ABB RAPID module: P901.mod

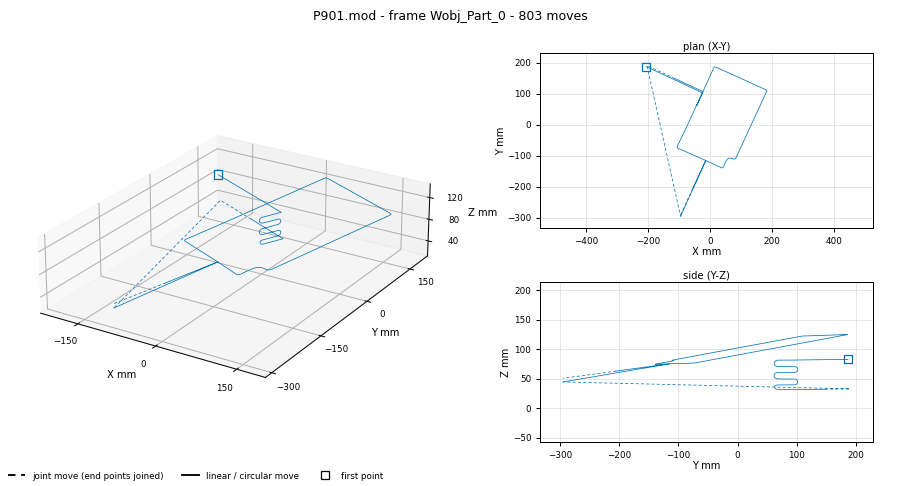
[picture p0: tool path of P901.mod in frame Wobj_Part_0, 803 of 813 moves have a stored position in this frame; points joined in program order, loops and branches not executed]
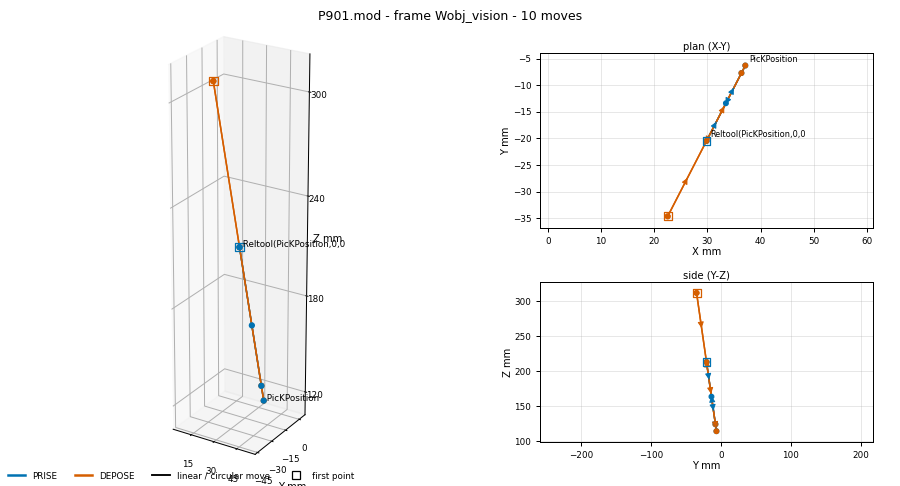
[picture p1: tool path of P901.mod in frame Wobj_vision, 10 of 813 moves have a stored position in this frame; points joined in program order, loops and branches not executed]
MODULE P901

    ! Nom         :P901
    ! Description :
    ! Créé le     :01/06/2023 14:08:14

    LOCAL CONST SPEEDDATA VitesseLente :=[3,500,0,0];
	LOCAL CONST SPEEDDATA VitesseRapide :=[30,500,0,0];
	LOCAL CONST SPEEDDATA VitesseTronconnage :=[2,500,0,0];
	LOCAL CONST SPEEDDATA VitesseTronconnageApp :=[10,500,0,0];
    !
    !Point de prise
    LOCAL PERS Robtarget PicKPosition := [[37.1247943324514,-6.27911838830437,114.674546951122],[0.0688762130874586,-0.531001244449083,0.843586238253387,0.0406940326553634],[0,0,0,0],[8.999999E+09,8.999999E+09,8.999999E+09,8.999999E+09,8.999999E+09,8.999999E+09]];
	LOCAL PERS Pose Ref := [[0,0,0],[1,0,0,0]];
    !
    !Declaration des points de meulage

    !Tr_meulage_motif_1 : Meulage d'un motif
    LOCAL CONST Robtarget Tr_meulage_motif_1_0 := [[-24.434275390625,103.0117734375,81.755546875],[0.378981302219628,-0.381323158247142,0.598057501703323,-0.594384594525059],[0,0,0,0],[8.999999E+09,8.999999E+09,8.999999E+09,8.999999E+09,8.999999E+09,8.999999E+09]];
    LOCAL CONST Robtarget Tr_meulage_motif_1_1 := [[-24.853365234375,102.103828125,81.7555625],[0.378981302219628,-0.381323158247142,0.598057501703323,-0.594384594525059],[0,0,0,0],[8.999999E+09,8.999999E+09,8.999999E+09,8.999999E+09,8.999999E+09,8.999999E+09]];
    LOCAL CONST Robtarget Tr_meulage_motif_1_2 := [[-25.27245703125,101.195890625,81.755578125],[0.378981302219628,-0.381323158247142,0.598057501703323,-0.594384594525059],[0,0,0,0],[8.999999E+09,8.999999E+09,8.999999E+09,8.999999E+09,8.999999E+09,8.999999E+09]];
    LOCAL CONST Robtarget Tr_meulage_motif_1_3 := [[-25.691546875,100.2879453125,81.75559375],[0.378981302219628,-0.381323158247142,0.598057501703323,-0.594384594525059],[0,0,0,0],[8.999999E+09,8.999999E+09,8.999999E+09,8.999999E+09,8.999999E+09,8.999999E+09]];
    LOCAL CONST Robtarget Tr_meulage_motif_1_4 := [[-26.11063671875,99.38,81.7556171875],[0.378981302219628,-0.381323158247142,0.598057501703323,-0.594384594525059],[0,0,0,0],[8.999999E+09,8.999999E+09,8.999999E+09,8.999999E+09,8.999999E+09,8.999999E+09]];
    LOCAL CONST Robtarget Tr_meulage_motif_1_5 := [[-26.5297265625,98.4720546875,81.7556328125],[0.378981302219628,-0.381323158247142,0.598057501703323,-0.594384594525059],[0,0,0,0],[8.999999E+09,8.999999E+09,8.999999E+09,8.999999E+09,8.999999E+09,8.999999E+09]];
    LOCAL CONST Robtarget Tr_meulage_motif_1_6 := [[-26.94881640625,97.564109375,81.7556484375],[0.378981302219628,-0.381323158247142,0.598057501703323,-0.594384594525059],[0,0,0,0],[8.999999E+09,8.999999E+09,8.999999E+09,8.999999E+09,8.999999E+09,8.999999E+09]];
    LOCAL CONST Robtarget Tr_meulage_motif_1_7 := [[-27.367908203125,96.6561640625,81.7556640625],[0.378981302219628,-0.381323158247142,0.598057501703323,-0.594384594525059],[0,0,0,0],[8.999999E+09,8.999999E+09,8.999999E+09,8.999999E+09,8.999999E+09,8.999999E+09]];
    LOCAL CONST Robtarget Tr_meulage_motif_1_8 := [[-27.786998046875,95.74821875,81.7556796875],[0.378981302219628,-0.381323158247142,0.598057501703323,-0.594384594525059],[0,0,0,0],[8.999999E+09,8.999999E+09,8.999999E+09,8.999999E+09,8.999999E+09,8.999999E+09]];
    LOCAL CONST Robtarget Tr_meulage_motif_1_9 := [[-28.206087890625,94.8402734375,81.7556953125],[0.378981302219628,-0.381323158247142,0.598057501703323,-0.594384594525059],[0,0,0,0],[8.999999E+09,8.999999E+09,8.999999E+09,8.999999E+09,8.999999E+09,8.999999E+09]];
    LOCAL CONST Robtarget Tr_meulage_motif_1_10 := [[-28.625177734375,93.932328125,81.7557109375],[0.378981302219628,-0.381323158247142,0.598057501703323,-0.594384594525059],[0,0,0,0],[8.999999E+09,8.999999E+09,8.999999E+09,8.999999E+09,8.999999E+09,8.999999E+09]];
    LOCAL CONST Robtarget Tr_meulage_motif_1_11 := [[-29.044267578125,93.0243828125,81.755734375],[0.378981302219628,-0.381323158247142,0.598057501703323,-0.594384594525059],[0,0,0,0],[8.999999E+09,8.999999E+09,8.999999E+09,8.999999E+09,8.999999E+09,8.999999E+09]];
    LOCAL CONST Robtarget Tr_meulage_motif_1_12 := [[-29.463359375,92.1164453125,81.75575],[0.378981302219628,-0.381323158247142,0.598057501703323,-0.594384594525059],[0,0,0,0],[8.999999E+09,8.999999E+09,8.999999E+09,8.999999E+09,8.999999E+09,8.999999E+09]];
    LOCAL CONST Robtarget Tr_meulage_motif_1_13 := [[-29.88244921875,91.2085,81.755765625],[0.378981302219628,-0.381323158247142,0.598057501703323,-0.594384594525059],[0,0,0,0],[8.999999E+09,8.999999E+09,8.999999E+09,8.999999E+09,8.999999E+09,8.999999E+09]];
    LOCAL CONST Robtarget Tr_meulage_motif_1_14 := [[-30.3015390625,90.3005546875,81.75578125],[0.378981302219628,-0.381323158247142,0.598057501703323,-0.594384594525059],[0,0,0,0],[8.999999E+09,8.999999E+09,8.999999E+09,8.999999E+09,8.999999E+09,8.999999E+09]];
    LOCAL CONST Robtarget Tr_meulage_motif_1_15 := [[-30.72062890625,89.392609375,81.755796875],[0.378981302219628,-0.381323158247142,0.598057501703323,-0.594384594525059],[0,0,0,0],[8.999999E+09,8.999999E+09,8.999999E+09,8.999999E+09,8.999999E+09,8.999999E+09]];
    LOCAL CONST Robtarget Tr_meulage_motif_1_16 := [[-31.13971875,88.4846640625,81.7558125],[0.378981302219628,-0.381323158247142,0.598057501703323,-0.594384594525059],[0,0,0,0],[8.999999E+09,8.999999E+09,8.999999E+09,8.999999E+09,8.999999E+09,8.999999E+09]];
    LOCAL CONST Robtarget Tr_meulage_motif_1_17 := [[-31.558810546875,87.57671875,81.755828125],[0.378981302219628,-0.381323158247142,0.598057501703323,-0.594384594525059],[0,0,0,0],[8.999999E+09,8.999999E+09,8.999999E+09,8.999999E+09,8.999999E+09,8.999999E+09]];
    LOCAL CONST Robtarget Tr_meulage_motif_1_18 := [[-31.977900390625,86.6687734375,81.7558515625],[0.378981302219628,-0.381323158247142,0.598057501703323,-0.594384594525059],[0,0,0,0],[8.999999E+09,8.999999E+09,8.999999E+09,8.999999E+09,8.999999E+09,8.999999E+09]];
    LOCAL CONST Robtarget Tr_meulage_motif_1_19 := [[-32.396990234375,85.760828125,81.7558671875],[0.378981302219628,-0.381323158247142,0.598057501703323,-0.594384594525059],[0,0,0,0],[8.999999E+09,8.999999E+09,8.999999E+09,8.999999E+09,8.999999E+09,8.999999E+09]];
    LOCAL CONST Robtarget Tr_meulage_motif_1_20 := [[-32.81608203125,84.8528828125,81.7558828125],[0.378981302219628,-0.381323158247142,0.598057501703323,-0.594384594525059],[0,0,0,0],[8.999999E+09,8.999999E+09,8.999999E+09,8.999999E+09,8.999999E+09,8.999999E+09]];
    LOCAL CONST Robtarget Tr_meulage_motif_1_21 := [[-33.235171875,83.9449375,81.7558984375],[0.378981302219628,-0.381323158247142,0.598057501703323,-0.594384594525059],[0,0,0,0],[8.999999E+09,8.999999E+09,8.999999E+09,8.999999E+09,8.999999E+09,8.999999E+09]];
    LOCAL CONST Robtarget Tr_meulage_motif_1_22 := [[-33.65426171875,83.0369921875,81.7559140625],[0.378981302219628,-0.381323158247142,0.598057501703323,-0.594384594525059],[0,0,0,0],[8.999999E+09,8.999999E+09,8.999999E+09,8.999999E+09,8.999999E+09,8.999999E+09]];
    LOCAL CONST Robtarget Tr_meulage_motif_1_23 := [[-34.0733515625,82.1290546875,81.7559296875],[0.378981302219628,-0.381323158247142,0.598057501703323,-0.594384594525059],[0,0,0,0],[8.999999E+09,8.999999E+09,8.999999E+09,8.999999E+09,8.999999E+09,8.999999E+09]];
    LOCAL CONST Robtarget Tr_meulage_motif_1_24 := [[-34.49244140625,81.221109375,81.755953125],[0.378981302219628,-0.381323158247142,0.598057501703323,-0.594384594525059],[0,0,0,0],[8.999999E+09,8.999999E+09,8.999999E+09,8.999999E+09,8.999999E+09,8.999999E+09]];
    LOCAL CONST Robtarget Tr_meulage_motif_1_25 := [[-34.91153125,80.3131640625,81.75596875],[0.378981302219628,-0.381323158247142,0.598057501703323,-0.594384594525059],[0,0,0,0],[8.999999E+09,8.999999E+09,8.999999E+09,8.999999E+09,8.999999E+09,8.999999E+09]];
    LOCAL CONST Robtarget Tr_meulage_motif_1_26 := [[-35.33062109375,79.40521875,81.755984375],[0.378981302219628,-0.381323158247142,0.598057501703323,-0.594384594525059],[0,0,0,0],[8.999999E+09,8.999999E+09,8.999999E+09,8.999999E+09,8.999999E+09,8.999999E+09]];
    LOCAL CONST Robtarget Tr_meulage_motif_1_27 := [[-35.7497109375,78.4972734375,81.756],[0.378981302219628,-0.381323158247142,0.598057501703323,-0.594384594525059],[0,0,0,0],[8.999999E+09,8.999999E+09,8.999999E+09,8.999999E+09,8.999999E+09,8.999999E+09]];
    LOCAL CONST Robtarget Tr_meulage_motif_1_28 := [[-36.16880078125,77.589328125,81.756015625],[0.378981302219628,-0.381323158247142,0.598057501703323,-0.594384594525059],[0,0,0,0],[8.999999E+09,8.999999E+09,8.999999E+09,8.999999E+09,8.999999E+09,8.999999E+09]];
    LOCAL CONST Robtarget Tr_meulage_motif_1_29 := [[-36.587890625,76.6813828125,81.75603125],[0.378981302219628,-0.381323158247142,0.598057501703323,-0.594384594525059],[0,0,0,0],[8.999999E+09,8.999999E+09,8.999999E+09,8.999999E+09,8.999999E+09,8.999999E+09]];
    LOCAL CONST Robtarget Tr_meulage_motif_1_30 := [[-37.006984375,75.7734375,81.756046875],[0.378981302219628,-0.381323158247142,0.598057501703323,-0.594384594525059],[0,0,0,0],[8.999999E+09,8.999999E+09,8.999999E+09,8.999999E+09,8.999999E+09,8.999999E+09]];
    LOCAL CONST Robtarget Tr_meulage_motif_1_31 := [[-37.42607421875,74.8654921875,81.7560703125],[0.378981302219628,-0.381323158247142,0.598057501703323,-0.594384594525059],[0,0,0,0],[8.999999E+09,8.999999E+09,8.999999E+09,8.999999E+09,8.999999E+09,8.999999E+09]];
    LOCAL CONST Robtarget Tr_meulage_motif_1_32 := [[-37.8451640625,73.957546875,81.7560859375],[0.378981302219628,-0.381323158247142,0.598057501703323,-0.594384594525059],[0,0,0,0],[8.999999E+09,8.999999E+09,8.999999E+09,8.999999E+09,8.999999E+09,8.999999E+09]];
    LOCAL CONST Robtarget Tr_meulage_motif_1_33 := [[-38.26425390625,73.0496015625,81.7561015625],[0.378981302219628,-0.381323158247142,0.598057501703323,-0.594384594525059],[0,0,0,0],[8.999999E+09,8.999999E+09,8.999999E+09,8.999999E+09,8.999999E+09,8.999999E+09]];
    LOCAL CONST Robtarget Tr_meulage_motif_1_34 := [[-38.68334375,72.1416640625,81.7561171875],[0.378981302219628,-0.381323158247142,0.598057501703323,-0.594384594525059],[0,0,0,0],[8.999999E+09,8.999999E+09,8.999999E+09,8.999999E+09,8.999999E+09,8.999999E+09]];
    LOCAL CONST Robtarget Tr_meulage_motif_1_35 := [[-39.10243359375,71.23371875,81.7561328125],[0.378981302219628,-0.381323158247142,0.598057501703323,-0.594384594525059],[0,0,0,0],[8.999999E+09,8.999999E+09,8.999999E+09,8.999999E+09,8.999999E+09,8.999999E+09]];
    LOCAL CONST Robtarget Tr_meulage_motif_1_36 := [[-39.5215234375,70.3257734375,81.7561484375],[0.378981302219628,-0.381323158247142,0.598057501703323,-0.594384594525059],[0,0,0,0],[8.999999E+09,8.999999E+09,8.999999E+09,8.999999E+09,8.999999E+09,8.999999E+09]];
    LOCAL CONST Robtarget Tr_meulage_motif_1_37 := [[-39.94061328125,69.417828125,81.7561640625],[0.378981302219628,-0.381323158247142,0.598057501703323,-0.594384594525059],[0,0,0,0],[8.999999E+09,8.999999E+09,8.999999E+09,8.999999E+09,8.999999E+09,8.999999E+09]];
    LOCAL CONST Robtarget Tr_meulage_motif_1_38 := [[-40.359703125,68.5098828125,81.7561875],[0.378981302219628,-0.381323158247142,0.598057501703323,-0.594384594525059],[0,0,0,0],[8.999999E+09,8.999999E+09,8.999999E+09,8.999999E+09,8.999999E+09,8.999999E+09]];
    LOCAL CONST Robtarget Tr_meulage_motif_1_39 := [[-40.77410546875,67.6079609375,81.6456171875],[0.378981302219628,-0.381323158247142,0.598057501703323,-0.594384594525059],[0,0,0,0],[8.999999E+09,8.999999E+09,8.999999E+09,8.999999E+09,8.999999E+09,8.999999E+09]];
    LOCAL CONST Robtarget Tr_meulage_motif_1_40 := [[-41.16776953125,66.747203125,81.4344765625],[0.378981302219628,-0.381323158247142,0.598057501703323,-0.594384594525059],[0,0,0,0],[8.999999E+09,8.999999E+09,8.999999E+09,8.999999E+09,8.999999E+09,8.999999E+09]];
    LOCAL CONST Robtarget Tr_meulage_motif_1_41 := [[-41.52126953125,65.9711953125,81.1626796875],[0.378981302219628,-0.381323158247142,0.598057501703323,-0.594384594525059],[0,0,0,0],[8.999999E+09,8.999999E+09,8.999999E+09,8.999999E+09,8.999999E+09,8.999999E+09]];
    LOCAL CONST Robtarget Tr_meulage_motif_1_42 := [[-41.83163671875,65.28847265625,80.8867890625],[0.378981302219628,-0.381323158247142,0.598057501703323,-0.594384594525059],[0,0,0,0],[8.999999E+09,8.999999E+09,8.999999E+09,8.999999E+09,8.999999E+09,8.999999E+09]];
    LOCAL CONST Robtarget Tr_meulage_motif_1_43 := [[-42.2843203125,64.28471484375,80.2707578125],[0.378981302219628,-0.381323158247142,0.598057501703323,-0.594384594525059],[0,0,0,0],[8.999999E+09,8.999999E+09,8.999999E+09,8.999999E+09,8.999999E+09,8.999999E+09]];
    LOCAL CONST Robtarget Tr_meulage_motif_1_44 := [[-42.701359375,63.34951171875,79.42321875],[0.378981302219628,-0.381323158247142,0.598057501703323,-0.594384594525059],[0,0,0,0],[8.999999E+09,8.999999E+09,8.999999E+09,8.999999E+09,8.999999E+09,8.999999E+09]];
    LOCAL CONST Robtarget Tr_meulage_motif_1_45 := [[-43.04204296875,62.5731484375,78.399484375],[0.378981302219628,-0.381323158247142,0.598057501703323,-0.594384594525059],[0,0,0,0],[8.999999E+09,8.999999E+09,8.999999E+09,8.999999E+09,8.999999E+09,8.999999E+09]];
    LOCAL CONST Robtarget Tr_meulage_motif_1_46 := [[-43.23075,62.122578125,77.2834453125],[0.378981302219628,-0.381323158247142,0.598057501703323,-0.594384594525059],[0,0,0,0],[8.999999E+09,8.999999E+09,8.999999E+09,8.999999E+09,8.999999E+09,8.999999E+09]];
    LOCAL CONST Robtarget Tr_meulage_motif_1_47 := [[-43.2321953125,62.09342578125,76.5875625],[0.378981302219628,-0.381323158247142,0.598057501703323,-0.594384594525059],[0,0,0,0],[8.999999E+09,8.999999E+09,8.999999E+09,8.999999E+09,8.999999E+09,8.999999E+09]];
    LOCAL CONST Robtarget Tr_meulage_motif_1_48 := [[-43.2227890625,62.08907421875,75.926390625],[0.378981302219628,-0.381323158247142,0.598057501703323,-0.594384594525059],[0,0,0,0],[8.999999E+09,8.999999E+09,8.999999E+09,8.999999E+09,8.999999E+09,8.999999E+09]];
    LOCAL CONST Robtarget Tr_meulage_motif_1_49 := [[-43.190390625,62.134546875,75.2653828125],[0.378981302219628,-0.381323158247142,0.598057501703323,-0.594384594525059],[0,0,0,0],[8.999999E+09,8.999999E+09,8.999999E+09,8.999999E+09,8.999999E+09,8.999999E+09]];
    LOCAL CONST Robtarget Tr_meulage_motif_1_50 := [[-42.965921875,62.5796484375,74.1637578125],[0.378981302219628,-0.381323158247142,0.598057501703323,-0.594384594525059],[0,0,0,0],[8.999999E+09,8.999999E+09,8.999999E+09,8.999999E+09,8.999999E+09,8.999999E+09]];
    LOCAL CONST Robtarget Tr_meulage_motif_1_51 := [[-42.59260546875,63.3507890625,73.1572421875],[0.378981302219628,-0.381323158247142,0.598057501703323,-0.594384594525059],[0,0,0,0],[8.999999E+09,8.999999E+09,8.999999E+09,8.999999E+09,8.999999E+09,8.999999E+09]];
    LOCAL CONST Robtarget Tr_meulage_motif_1_52 := [[-42.15191796875,64.27452734375,72.328453125],[0.378981302219628,-0.381323158247142,0.598057501703323,-0.594384594525059],[0,0,0,0],[8.999999E+09,8.999999E+09,8.999999E+09,8.999999E+09,8.999999E+09,8.999999E+09]];
    LOCAL CONST Robtarget Tr_meulage_motif_1_53 := [[-41.85833203125,64.895765625,71.932734375],[0.378981302219628,-0.381323158247142,0.598057501703323,-0.594384594525059],[0,0,0,0],[8.999999E+09,8.999999E+09,8.999999E+09,8.999999E+09,8.999999E+09,8.999999E+09]];
    LOCAL CONST Robtarget Tr_meulage_motif_1_54 := [[-41.36602734375,65.9441015625,71.44525],[0.378981302219628,-0.381323158247142,0.598057501703323,-0.594384594525059],[0,0,0,0],[8.999999E+09,8.999999E+09,8.999999E+09,8.999999E+09,8.999999E+09,8.999999E+09]];
    LOCAL CONST Robtarget Tr_meulage_motif_1_55 := [[-41.00812890625,66.7096015625,71.181171875],[0.378981302219628,-0.381323158247142,0.598057501703323,-0.594384594525059],[0,0,0,0],[8.999999E+09,8.999999E+09,8.999999E+09,8.999999E+09,8.999999E+09,8.999999E+09]];
    LOCAL CONST Robtarget Tr_meulage_motif_1_56 := [[-40.61462890625,67.5544609375,70.9767109375],[0.378981302219628,-0.381323158247142,0.598057501703323,-0.594384594525059],[0,0,0,0],[8.999999E+09,8.999999E+09,8.999999E+09,8.999999E+09,8.999999E+09,8.999999E+09]];
    LOCAL CONST Robtarget Tr_meulage_motif_1_57 := [[-40.20171875,68.444953125,70.8681171875],[0.378981302219628,-0.381323158247142,0.598057501703323,-0.594384594525059],[0,0,0,0],[8.999999E+09,8.999999E+09,8.999999E+09,8.999999E+09,8.999999E+09,8.999999E+09]];
    LOCAL CONST Robtarget Tr_meulage_motif_1_58 := [[-39.78417578125,69.3454140625,70.757515625],[0.378981302219628,-0.381323158247142,0.598057501703323,-0.594384594525059],[0,0,0,0],[8.999999E+09,8.999999E+09,8.999999E+09,8.999999E+09,8.999999E+09,8.999999E+09]];
    LOCAL CONST Robtarget Tr_meulage_motif_1_59 := [[-39.3650859375,70.253359375,70.7575],[0.378981302219628,-0.381323158247142,0.598057501703323,-0.594384594525059],[0,0,0,0],[8.999999E+09,8.999999E+09,8.999999E+09,8.999999E+09,8.999999E+09,8.999999E+09]];
    LOCAL CONST Robtarget Tr_meulage_motif_1_60 := [[-38.9459921875,71.1613046875,70.757484375],[0.378981302219628,-0.381323158247142,0.598057501703323,-0.594384594525059],[0,0,0,0],[8.999999E+09,8.999999E+09,8.999999E+09,8.999999E+09,8.999999E+09,8.999999E+09]];
    LOCAL CONST Robtarget Tr_meulage_motif_1_61 := [[-38.52690234375,72.06925,70.75746875],[0.378981302219628,-0.381323158247142,0.598057501703323,-0.594384594525059],[0,0,0,0],[8.999999E+09,8.999999E+09,8.999999E+09,8.999999E+09,8.999999E+09,8.999999E+09]];
    LOCAL CONST Robtarget Tr_meulage_motif_1_62 := [[-38.1078125,72.9771953125,70.757453125],[0.378981302219628,-0.381323158247142,0.598057501703323,-0.594384594525059],[0,0,0,0],[8.999999E+09,8.999999E+09,8.999999E+09,8.999999E+09,8.999999E+09,8.999999E+09]];
    LOCAL CONST Robtarget Tr_meulage_motif_1_63 := [[-37.68872265625,73.8851328125,70.7574375],[0.378981302219628,-0.381323158247142,0.598057501703323,-0.594384594525059],[0,0,0,0],[8.999999E+09,8.999999E+09,8.999999E+09,8.999999E+09,8.999999E+09,8.999999E+09]];
    LOCAL CONST Robtarget Tr_meulage_motif_1_64 := [[-37.2696328125,74.793078125,70.7574140625],[0.378981302219628,-0.381323158247142,0.598057501703323,-0.594384594525059],[0,0,0,0],[8.999999E+09,8.999999E+09,8.999999E+09,8.999999E+09,8.999999E+09,8.999999E+09]];
    LOCAL CONST Robtarget Tr_meulage_motif_1_65 := [[-36.85054296875,75.7010234375,70.7573984375],[0.378981302219628,-0.381323158247142,0.598057501703323,-0.594384594525059],[0,0,0,0],[8.999999E+09,8.999999E+09,8.999999E+09,8.999999E+09,8.999999E+09,8.999999E+09]];
    LOCAL CONST Robtarget Tr_meulage_motif_1_66 := [[-36.431453125,76.60896875,70.7573828125],[0.378981302219628,-0.381323158247142,0.598057501703323,-0.594384594525059],[0,0,0,0],[8.999999E+09,8.999999E+09,8.999999E+09,8.999999E+09,8.999999E+09,8.999999E+09]];
    LOCAL CONST Robtarget Tr_meulage_motif_1_67 := [[-36.01236328125,77.5169140625,70.7573671875],[0.378981302219628,-0.381323158247142,0.598057501703323,-0.594384594525059],[0,0,0,0],[8.999999E+09,8.999999E+09,8.999999E+09,8.999999E+09,8.999999E+09,8.999999E+09]];
    LOCAL CONST Robtarget Tr_meulage_motif_1_68 := [[-35.5932734375,78.424859375,70.7573515625],[0.378981302219628,-0.381323158247142,0.598057501703323,-0.594384594525059],[0,0,0,0],[8.999999E+09,8.999999E+09,8.999999E+09,8.999999E+09,8.999999E+09,8.999999E+09]];
    LOCAL CONST Robtarget Tr_meulage_motif_1_69 := [[-35.17418359375,79.3328046875,70.7573359375],[0.378981302219628,-0.381323158247142,0.598057501703323,-0.594384594525059],[0,0,0,0],[8.999999E+09,8.999999E+09,8.999999E+09,8.999999E+09,8.999999E+09,8.999999E+09]];
    LOCAL CONST Robtarget Tr_meulage_motif_1_70 := [[-34.75508984375,80.24075,70.7573203125],[0.378981302219628,-0.381323158247142,0.598057501703323,-0.594384594525059],[0,0,0,0],[8.999999E+09,8.999999E+09,8.999999E+09,8.999999E+09,8.999999E+09,8.999999E+09]];
    LOCAL CONST Robtarget Tr_meulage_motif_1_71 := [[-34.336,81.1486953125,70.757296875],[0.378981302219628,-0.381323158247142,0.598057501703323,-0.594384594525059],[0,0,0,0],[8.999999E+09,8.999999E+09,8.999999E+09,8.999999E+09,8.999999E+09,8.999999E+09]];
    LOCAL CONST Robtarget Tr_meulage_motif_1_72 := [[-33.91691015625,82.056640625,70.75728125],[0.378981302219628,-0.381323158247142,0.598057501703323,-0.594384594525059],[0,0,0,0],[8.999999E+09,8.999999E+09,8.999999E+09,8.999999E+09,8.999999E+09,8.999999E+09]];
    LOCAL CONST Robtarget Tr_meulage_motif_1_73 := [[-33.4978203125,82.9645859375,70.757265625],[0.378981302219628,-0.381323158247142,0.598057501703323,-0.594384594525059],[0,0,0,0],[8.999999E+09,8.999999E+09,8.999999E+09,8.999999E+09,8.999999E+09,8.999999E+09]];
    LOCAL CONST Robtarget Tr_meulage_motif_1_74 := [[-33.07873046875,83.8725234375,70.75725],[0.378981302219628,-0.381323158247142,0.598057501703323,-0.594384594525059],[0,0,0,0],[8.999999E+09,8.999999E+09,8.999999E+09,8.999999E+09,8.999999E+09,8.999999E+09]];
    LOCAL CONST Robtarget Tr_meulage_motif_1_75 := [[-32.659640625,84.78046875,70.757234375],[0.378981302219628,-0.381323158247142,0.598057501703323,-0.594384594525059],[0,0,0,0],[8.999999E+09,8.999999E+09,8.999999E+09,8.999999E+09,8.999999E+09,8.999999E+09]];
    LOCAL CONST Robtarget Tr_meulage_motif_1_76 := [[-32.24055078125,85.6884140625,70.75721875],[0.378981302219628,-0.381323158247142,0.598057501703323,-0.594384594525059],[0,0,0,0],[8.999999E+09,8.999999E+09,8.999999E+09,8.999999E+09,8.999999E+09,8.999999E+09]];
    LOCAL CONST Robtarget Tr_meulage_motif_1_77 := [[-31.821458984375,86.596359375,70.757203125],[0.378981302219628,-0.381323158247142,0.598057501703323,-0.594384594525059],[0,0,0,0],[8.999999E+09,8.999999E+09,8.999999E+09,8.999999E+09,8.999999E+09,8.999999E+09]];
    LOCAL CONST Robtarget Tr_meulage_motif_1_78 := [[-31.402369140625,87.5043046875,70.7571796875],[0.378981302219628,-0.381323158247142,0.598057501703323,-0.594384594525059],[0,0,0,0],[8.999999E+09,8.999999E+09,8.999999E+09,8.999999E+09,8.999999E+09,8.999999E+09]];
    LOCAL CONST Robtarget Tr_meulage_motif_1_79 := [[-30.983279296875,88.41225,70.7571640625],[0.378981302219628,-0.381323158247142,0.598057501703323,-0.594384594525059],[0,0,0,0],[8.999999E+09,8.999999E+09,8.999999E+09,8.999999E+09,8.999999E+09,8.999999E+09]];
    LOCAL CONST Robtarget Tr_meulage_motif_1_80 := [[-30.564189453125,89.3201953125,70.7571484375],[0.378981302219628,-0.381323158247142,0.598057501703323,-0.594384594525059],[0,0,0,0],[8.999999E+09,8.999999E+09,8.999999E+09,8.999999E+09,8.999999E+09,8.999999E+09]];
    LOCAL CONST Robtarget Tr_meulage_motif_1_81 := [[-30.145099609375,90.228140625,70.7571328125],[0.378981302219628,-0.381323158247142,0.598057501703323,-0.594384594525059],[0,0,0,0],[8.999999E+09,8.999999E+09,8.999999E+09,8.999999E+09,8.999999E+09,8.999999E+09]];
    LOCAL CONST Robtarget Tr_meulage_motif_1_82 := [[-29.7260078125,91.1360859375,70.7571171875],[0.378981302219628,-0.381323158247142,0.598057501703323,-0.594384594525059],[0,0,0,0],[8.999999E+09,8.999999E+09,8.999999E+09,8.999999E+09,8.999999E+09,8.999999E+09]];
    LOCAL CONST Robtarget Tr_meulage_motif_1_83 := [[-29.30691796875,92.04403125,70.7571015625],[0.378981302219628,-0.381323158247142,0.598057501703323,-0.594384594525059],[0,0,0,0],[8.999999E+09,8.999999E+09,8.999999E+09,8.999999E+09,8.999999E+09,8.999999E+09]];
    LOCAL CONST Robtarget Tr_meulage_motif_1_84 := [[-28.887828125,92.9519765625,70.7570859375],[0.378981302219628,-0.381323158247142,0.598057501703323,-0.594384594525059],[0,0,0,0],[8.999999E+09,8.999999E+09,8.999999E+09,8.999999E+09,8.999999E+09,8.999999E+09]];
    LOCAL CONST Robtarget Tr_meulage_motif_1_85 := [[-28.46873828125,93.8599140625,70.7570625],[0.378981302219628,-0.381323158247142,0.598057501703323,-0.594384594525059],[0,0,0,0],[8.999999E+09,8.999999E+09,8.999999E+09,8.999999E+09,8.999999E+09,8.999999E+09]];
    LOCAL CONST Robtarget Tr_meulage_motif_1_86 := [[-28.0496484375,94.767859375,70.757046875],[0.378981302219628,-0.381323158247142,0.598057501703323,-0.594384594525059],[0,0,0,0],[8.999999E+09,8.999999E+09,8.999999E+09,8.999999E+09,8.999999E+09,8.999999E+09]];
    LOCAL CONST Robtarget Tr_meulage_motif_1_87 := [[-27.63055859375,95.6758046875,70.75703125],[0.378981302219628,-0.381323158247142,0.598057501703323,-0.594384594525059],[0,0,0,0],[8.999999E+09,8.999999E+09,8.999999E+09,8.999999E+09,8.999999E+09,8.999999E+09]];
    LOCAL CONST Robtarget Tr_meulage_motif_1_88 := [[-27.211466796875,96.58375,70.757015625],[0.378981302219628,-0.381323158247142,0.598057501703323,-0.594384594525059],[0,0,0,0],[8.999999E+09,8.999999E+09,8.999999E+09,8.999999E+09,8.999999E+09,8.999999E+09]];
    LOCAL CONST Robtarget Tr_meulage_motif_1_89 := [[-26.793921875,97.48421875,70.646421875],[0.378981302219628,-0.381323158247142,0.598057501703323,-0.594384594525059],[0,0,0,0],[8.999999E+09,8.999999E+09,8.999999E+09,8.999999E+09,8.999999E+09,8.999999E+09]];
    LOCAL CONST Robtarget Tr_meulage_motif_1_90 := [[-26.394248046875,98.3421953125,70.4352421875],[0.378981302219628,-0.381323158247142,0.598057501703323,-0.594384594525059],[0,0,0,0],[8.999999E+09,8.999999E+09,8.999999E+09,8.999999E+09,8.999999E+09,8.999999E+09]];
    LOCAL CONST Robtarget Tr_meulage_motif_1_91 := [[-26.033017578125,99.114625,70.1634140625],[0.378981302219628,-0.381323158247142,0.598057501703323,-0.594384594525059],[0,0,0,0],[8.999999E+09,8.999999E+09,8.999999E+09,8.999999E+09,8.999999E+09,8.999999E+09]];
    LOCAL CONST Robtarget Tr_meulage_motif_1_92 := [[-25.7305078125,99.758625,69.8592890625],[0.378981302219628,-0.381323158247142,0.598057501703323,-0.594384594525059],[0,0,0,0],[8.999999E+09,8.999999E+09,8.999999E+09,8.999999E+09,8.999999E+09,8.999999E+09]];
    LOCAL CONST Robtarget Tr_meulage_motif_1_93 := [[-25.28755078125,100.6935078125,69.1968203125],[0.378981302219628,-0.381323158247142,0.598057501703323,-0.594384594525059],[0,0,0,0],[8.999999E+09,8.999999E+09,8.999999E+09,8.999999E+09,8.999999E+09,8.999999E+09]];
    LOCAL CONST Robtarget Tr_meulage_motif_1_94 := [[-24.89673046875,101.5064765625,68.2949765625],[0.378981302219628,-0.381323158247142,0.598057501703323,-0.594384594525059],[0,0,0,0],[8.999999E+09,8.999999E+09,8.999999E+09,8.999999E+09,8.999999E+09,8.999999E+09]];
    LOCAL CONST Robtarget Tr_meulage_motif_1_95 := [[-24.65765234375,101.9853125,67.2490625],[0.378981302219628,-0.381323158247142,0.598057501703323,-0.594384594525059],[0,0,0,0],[8.999999E+09,8.999999E+09,8.999999E+09,8.999999E+09,8.999999E+09,8.999999E+09]];
    LOCAL CONST Robtarget Tr_meulage_motif_1_96 := [[-24.570353515625,102.1485234375,66.5559296875],[0.378981302219628,-0.381323158247142,0.598057501703323,-0.594384594525059],[0,0,0,0],[8.999999E+09,8.999999E+09,8.999999E+09,8.999999E+09,8.999999E+09,8.999999E+09]];
    LOCAL CONST Robtarget Tr_meulage_motif_1_97 := [[-24.532646484375,102.201421875,65.7860234375],[0.378981302219628,-0.381323158247142,0.598057501703323,-0.594384594525059],[0,0,0,0],[8.999999E+09,8.999999E+09,8.999999E+09,8.999999E+09,8.999999E+09,8.999999E+09]];
    LOCAL CONST Robtarget Tr_meulage_motif_1_98 := [[-24.549751953125,102.135578125,65.0162421875],[0.378981302219628,-0.381323158247142,0.598057501703323,-0.594384594525059],[0,0,0,0],[8.999999E+09,8.999999E+09,8.999999E+09,8.999999E+09,8.999999E+09,8.999999E+09]];
    LOCAL CONST Robtarget Tr_meulage_motif_1_99 := [[-24.709837890625,101.7473125,63.90813671875],[0.378981302219628,-0.381323158247142,0.598057501703323,-0.594384594525059],[0,0,0,0],[8.999999E+09,8.999999E+09,8.999999E+09,8.999999E+09,8.999999E+09,8.999999E+09]];
    LOCAL CONST Robtarget Tr_meulage_motif_1_100 := [[-24.875142578125,101.36728125,63.32252734375],[0.378981302219628,-0.381323158247142,0.598057501703323,-0.594384594525059],[0,0,0,0],[8.999999E+09,8.999999E+09,8.999999E+09,8.999999E+09,8.999999E+09,8.999999E+09]];
    LOCAL CONST Robtarget Tr_meulage_motif_1_101 := [[-25.234310546875,100.555984375,62.4355234375],[0.378981302219628,-0.381323158247142,0.598057501703323,-0.594384594525059],[0,0,0,0],[8.999999E+09,8.999999E+09,8.999999E+09,8.999999E+09,8.999999E+09,8.999999E+09]];
    LOCAL CONST Robtarget Tr_meulage_motif_1_102 := [[-25.473875,100.021484375,62.0212734375],[0.378981302219628,-0.381323158247142,0.598057501703323,-0.594384594525059],[0,0,0,0],[8.999999E+09,8.999999E+09,8.999999E+09,8.999999E+09,8.999999E+09,8.999999E+09]];
    LOCAL CONST Robtarget Tr_meulage_motif_1_103 := [[-25.934640625,99.00290625,61.477265625],[0.378981302219628,-0.381323158247142,0.598057501703323,-0.594384594525059],[0,0,0,0],[8.999999E+09,8.999999E+09,8.999999E+09,8.999999E+09,8.999999E+09,8.999999E+09]];
    LOCAL CONST Robtarget Tr_meulage_motif_1_104 := [[-26.276435546875,98.2513671875,61.18181640625],[0.378981302219628,-0.381323158247142,0.598057501703323,-0.594384594525059],[0,0,0,0],[8.999999E+09,8.999999E+09,8.999999E+09,8.999999E+09,8.999999E+09,8.999999E+09]];
    LOCAL CONST Robtarget Tr_meulage_motif_1_105 := [[-26.66412109375,97.4038125,60.97738671875],[0.378981302219628,-0.381323158247142,0.598057501703323,-0.594384594525059],[0,0,0,0],[8.999999E+09,8.999999E+09,8.999999E+09,8.999999E+09,8.999999E+09,8.999999E+09]];
    LOCAL CONST Robtarget Tr_meulage_motif_1_106 := [[-27.073939453125,96.5118984375,60.86882421875],[0.378981302219628,-0.381323158247142,0.598057501703323,-0.594384594525059],[0,0,0,0],[8.999999E+09,8.999999E+09,8.999999E+09,8.999999E+09,8.999999E+09,8.999999E+09]];
    LOCAL CONST Robtarget Tr_meulage_motif_1_107 := [[-27.48833984375,95.6099765625,60.7582578125],[0.378981302219628,-0.381323158247142,0.598057501703323,-0.594384594525059],[0,0,0,0],[8.999999E+09,8.999999E+09,8.999999E+09,8.999999E+09,8.999999E+09,8.999999E+09]];
    LOCAL CONST Robtarget Tr_meulage_motif_1_108 := [[-27.9074296875,94.70203125,60.75827734375],[0.378981302219628,-0.381323158247142,0.598057501703323,-0.594384594525059],[0,0,0,0],[8.999999E+09,8.999999E+09,8.999999E+09,8.999999E+09,8.999999E+09,8.999999E+09]];
    LOCAL CONST Robtarget Tr_meulage_motif_1_109 := [[-28.32651953125,93.7940859375,60.75829296875],[0.378981302219628,-0.381323158247142,0.598057501703323,-0.594384594525059],[0,0,0,0],[8.999999E+09,8.999999E+09,8.999999E+09,8.999999E+09,8.999999E+09,8.999999E+09]];
    LOCAL CONST Robtarget Tr_meulage_motif_1_110 := [[-28.745609375,92.886140625,60.75830859375],[0.378981302219628,-0.381323158247142,0.598057501703323,-0.594384594525059],[0,0,0,0],[8.999999E+09,8.999999E+09,8.999999E+09,8.999999E+09,8.999999E+09,8.999999E+09]];
    LOCAL CONST Robtarget Tr_meulage_motif_1_111 := [[-29.164701171875,91.9781953125,60.758328125],[0.378981302219628,-0.381323158247142,0.598057501703323,-0.594384594525059],[0,0,0,0],[8.999999E+09,8.999999E+09,8.999999E+09,8.999999E+09,8.999999E+09,8.999999E+09]];
    LOCAL CONST Robtarget Tr_meulage_motif_1_112 := [[-29.583791015625,91.0702578125,60.75834375],[0.378981302219628,-0.381323158247142,0.598057501703323,-0.594384594525059],[0,0,0,0],[8.999999E+09,8.999999E+09,8.999999E+09,8.999999E+09,8.999999E+09,8.999999E+09]];
    LOCAL CONST Robtarget Tr_meulage_motif_1_113 := [[-30.002880859375,90.1623125,60.758359375],[0.378981302219628,-0.381323158247142,0.598057501703323,-0.594384594525059],[0,0,0,0],[8.999999E+09,8.999999E+09,8.999999E+09,8.999999E+09,8.999999E+09,8.999999E+09]];
    LOCAL CONST Robtarget Tr_meulage_motif_1_114 := [[-30.421970703125,89.2543671875,60.75837890625],[0.378981302219628,-0.381323158247142,0.598057501703323,-0.594384594525059],[0,0,0,0],[8.999999E+09,8.999999E+09,8.999999E+09,8.999999E+09,8.999999E+09,8.999999E+09]];
    LOCAL CONST Robtarget Tr_meulage_motif_1_115 := [[-30.841060546875,88.346421875,60.75839453125],[0.378981302219628,-0.381323158247142,0.598057501703323,-0.594384594525059],[0,0,0,0],[8.999999E+09,8.999999E+09,8.999999E+09,8.999999E+09,8.999999E+09,8.999999E+09]];
    LOCAL CONST Robtarget Tr_meulage_motif_1_116 := [[-31.26015234375,87.4384765625,60.75841015625],[0.378981302219628,-0.381323158247142,0.598057501703323,-0.594384594525059],[0,0,0,0],[8.999999E+09,8.999999E+09,8.999999E+09,8.999999E+09,8.999999E+09,8.999999E+09]];
    LOCAL CONST Robtarget Tr_meulage_motif_1_117 := [[-31.6792421875,86.53053125,60.75842578125],[0.378981302219628,-0.381323158247142,0.598057501703323,-0.594384594525059],[0,0,0,0],[8.999999E+09,8.999999E+09,8.999999E+09,8.999999E+09,8.999999E+09,8.999999E+09]];
    LOCAL CONST Robtarget Tr_meulage_motif_1_118 := [[-32.09833203125,85.6225859375,60.7584453125],[0.378981302219628,-0.381323158247142,0.598057501703323,-0.594384594525059],[0,0,0,0],[8.999999E+09,8.999999E+09,8.999999E+09,8.999999E+09,8.999999E+09,8.999999E+09]];
    LOCAL CONST Robtarget Tr_meulage_motif_1_119 := [[-32.517421875,84.714640625,60.7584609375],[0.378981302219628,-0.381323158247142,0.598057501703323,-0.594384594525059],[0,0,0,0],[8.999999E+09,8.999999E+09,8.999999E+09,8.999999E+09,8.999999E+09,8.999999E+09]];
    LOCAL CONST Robtarget Tr_meulage_motif_1_120 := [[-32.93651171875,83.8066953125,60.7584765625],[0.378981302219628,-0.381323158247142,0.598057501703323,-0.594384594525059],[0,0,0,0],[8.999999E+09,8.999999E+09,8.999999E+09,8.999999E+09,8.999999E+09,8.999999E+09]];
    LOCAL CONST Robtarget Tr_meulage_motif_1_121 := [[-33.3556015625,82.89875,60.75849609375],[0.378981302219628,-0.381323158247142,0.598057501703323,-0.594384594525059],[0,0,0,0],[8.999999E+09,8.999999E+09,8.999999E+09,8.999999E+09,8.999999E+09,8.999999E+09]];
    LOCAL CONST Robtarget Tr_meulage_motif_1_122 := [[-33.77469140625,81.9908046875,60.75851171875],[0.378981302219628,-0.381323158247142,0.598057501703323,-0.594384594525059],[0,0,0,0],[8.999999E+09,8.999999E+09,8.999999E+09,8.999999E+09,8.999999E+09,8.999999E+09]];
    LOCAL CONST Robtarget Tr_meulage_motif_1_123 := [[-34.19378125,81.0828671875,60.75852734375],[0.378981302219628,-0.381323158247142,0.598057501703323,-0.594384594525059],[0,0,0,0],[8.999999E+09,8.999999E+09,8.999999E+09,8.999999E+09,8.999999E+09,8.999999E+09]];
    LOCAL CONST Robtarget Tr_meulage_motif_1_124 := [[-34.612875,80.174921875,60.758546875],[0.378981302219628,-0.381323158247142,0.598057501703323,-0.594384594525059],[0,0,0,0],[8.999999E+09,8.999999E+09,8.999999E+09,8.999999E+09,8.999999E+09,8.999999E+09]];
    LOCAL CONST Robtarget Tr_meulage_motif_1_125 := [[-35.03196484375,79.2669765625,60.7585625],[0.378981302219628,-0.381323158247142,0.598057501703323,-0.594384594525059],[0,0,0,0],[8.999999E+09,8.999999E+09,8.999999E+09,8.999999E+09,8.999999E+09,8.999999E+09]];
    LOCAL CONST Robtarget Tr_meulage_motif_1_126 := [[-35.4510546875,78.35903125,60.758578125],[0.378981302219628,-0.381323158247142,0.598057501703323,-0.594384594525059],[0,0,0,0],[8.999999E+09,8.999999E+09,8.999999E+09,8.999999E+09,8.999999E+09,8.999999E+09]];
    LOCAL CONST Robtarget Tr_meulage_motif_1_127 := [[-35.87014453125,77.4510859375,60.75859375],[0.378981302219628,-0.381323158247142,0.598057501703323,-0.594384594525059],[0,0,0,0],[8.999999E+09,8.999999E+09,8.999999E+09,8.999999E+09,8.999999E+09,8.999999E+09]];
    LOCAL CONST Robtarget Tr_meulage_motif_1_128 := [[-36.289234375,76.543140625,60.75861328125],[0.378981302219628,-0.381323158247142,0.598057501703323,-0.594384594525059],[0,0,0,0],[8.999999E+09,8.999999E+09,8.999999E+09,8.999999E+09,8.999999E+09,8.999999E+09]];
    LOCAL CONST Robtarget Tr_meulage_motif_1_129 := [[-36.70832421875,75.6351953125,60.75862890625],[0.378981302219628,-0.381323158247142,0.598057501703323,-0.594384594525059],[0,0,0,0],[8.999999E+09,8.999999E+09,8.999999E+09,8.999999E+09,8.999999E+09,8.999999E+09]];
    LOCAL CONST Robtarget Tr_meulage_motif_1_130 := [[-37.1274140625,74.72725,60.75864453125],[0.378981302219628,-0.381323158247142,0.598057501703323,-0.594384594525059],[0,0,0,0],[8.999999E+09,8.999999E+09,8.999999E+09,8.999999E+09,8.999999E+09,8.999999E+09]];
    LOCAL CONST Robtarget Tr_meulage_motif_1_131 := [[-37.54650390625,73.8193046875,60.7586640625],[0.378981302219628,-0.381323158247142,0.598057501703323,-0.594384594525059],[0,0,0,0],[8.999999E+09,8.999999E+09,8.999999E+09,8.999999E+09,8.999999E+09,8.999999E+09]];
    LOCAL CONST Robtarget Tr_meulage_motif_1_132 := [[-37.96559375,72.911359375,60.7586796875],[0.378981302219628,-0.381323158247142,0.598057501703323,-0.594384594525059],[0,0,0,0],[8.999999E+09,8.999999E+09,8.999999E+09,8.999999E+09,8.999999E+09,8.999999E+09]];
    LOCAL CONST Robtarget Tr_meulage_motif_1_133 := [[-38.38468359375,72.0034140625,60.7586953125],[0.378981302219628,-0.381323158247142,0.598057501703323,-0.594384594525059],[0,0,0,0],[8.999999E+09,8.999999E+09,8.999999E+09,8.999999E+09,8.999999E+09,8.999999E+09]];
    LOCAL CONST Robtarget Tr_meulage_motif_1_134 := [[-38.80377734375,71.0954765625,60.7587109375],[0.378981302219628,-0.381323158247142,0.598057501703323,-0.594384594525059],[0,0,0,0],[8.999999E+09,8.999999E+09,8.999999E+09,8.999999E+09,8.999999E+09,8.999999E+09]];
    LOCAL CONST Robtarget Tr_meulage_motif_1_135 := [[-39.2228671875,70.18753125,60.75873046875],[0.378981302219628,-0.381323158247142,0.598057501703323,-0.594384594525059],[0,0,0,0],[8.999999E+09,8.999999E+09,8.999999E+09,8.999999E+09,8.999999E+09,8.999999E+09]];
    LOCAL CONST Robtarget Tr_meulage_motif_1_136 := [[-39.64195703125,69.2795859375,60.75874609375],[0.378981302219628,-0.381323158247142,0.598057501703323,-0.594384594525059],[0,0,0,0],[8.999999E+09,8.999999E+09,8.999999E+09,8.999999E+09,8.999999E+09,8.999999E+09]];
    LOCAL CONST Robtarget Tr_meulage_motif_1_137 := [[-40.061046875,68.371640625,60.75876171875],[0.378981302219628,-0.381323158247142,0.598057501703323,-0.594384594525059],[0,0,0,0],[8.999999E+09,8.999999E+09,8.999999E+09,8.999999E+09,8.999999E+09,8.999999E+09]];
    LOCAL CONST Robtarget Tr_meulage_motif_1_138 := [[-40.4754453125,67.46971875,60.64819921875],[0.378981302219628,-0.381323158247142,0.598057501703323,-0.594384594525059],[0,0,0,0],[8.999999E+09,8.999999E+09,8.999999E+09,8.999999E+09,8.999999E+09,8.999999E+09]];
    LOCAL CONST Robtarget Tr_meulage_motif_1_139 := [[-40.86911328125,66.6089609375,60.4370546875],[0.378981302219628,-0.381323158247142,0.598057501703323,-0.594384594525059],[0,0,0,0],[8.999999E+09,8.999999E+09,8.999999E+09,8.999999E+09,8.999999E+09,8.999999E+09]];
    LOCAL CONST Robtarget Tr_meulage_motif_1_140 := [[-41.22261328125,65.8329453125,60.1652578125],[0.378981302219628,-0.381323158247142,0.598057501703323,-0.594384594525059],[0,0,0,0],[8.999999E+09,8.999999E+09,8.999999E+09,8.999999E+09,8.999999E+09,8.999999E+09]];
    LOCAL CONST Robtarget Tr_meulage_motif_1_141 := [[-41.53298046875,65.15023046875,59.8893671875],[0.378981302219628,-0.381323158247142,0.598057501703323,-0.594384594525059],[0,0,0,0],[8.999999E+09,8.999999E+09,8.999999E+09,8.999999E+09,8.999999E+09,8.999999E+09]];
    LOCAL CONST Robtarget Tr_meulage_motif_1_142 := [[-41.98566015625,64.14647265625,59.2733359375],[0.378981302219628,-0.381323158247142,0.598057501703323,-0.594384594525059],[0,0,0,0],[8.999999E+09,8.999999E+09,8.999999E+09,8.999999E+09,8.999999E+09,8.999999E+09]];
    LOCAL CONST Robtarget Tr_meulage_motif_1_143 := [[-42.402703125,63.21126953125,58.42580078125],[0.378981302219628,-0.381323158247142,0.598057501703323,-0.594384594525059],[0,0,0,0],[8.999999E+09,8.999999E+09,8.999999E+09,8.999999E+09,8.999999E+09,8.999999E+09]];
    LOCAL CONST Robtarget Tr_meulage_motif_1_144 := [[-42.74338671875,62.43490234375,57.40206640625],[0.378981302219628,-0.381323158247142,0.598057501703323,-0.594384594525059],[0,0,0,0],[8.999999E+09,8.999999E+09,8.999999E+09,8.999999E+09,8.999999E+09,8.999999E+09]];
    LOCAL CONST Robtarget Tr_meulage_motif_1_145 := [[-42.93209375,61.9843359375,56.2860234375],[0.378981302219628,-0.381323158247142,0.598057501703323,-0.594384594525059],[0,0,0,0],[8.999999E+09,8.999999E+09,8.999999E+09,8.999999E+09,8.999999E+09,8.999999E+09]];
    LOCAL CONST Robtarget Tr_meulage_motif_1_146 := [[-42.93353515625,61.95518359375,55.590140625],[0.378981302219628,-0.381323158247142,0.598057501703323,-0.594384594525059],[0,0,0,0],[8.999999E+09,8.999999E+09,8.999999E+09,8.999999E+09,8.999999E+09,8.999999E+09]];
    LOCAL CONST Robtarget Tr_meulage_motif_1_147 := [[-42.9241328125,61.95083203125,54.92897265625],[0.378981302219628,-0.381323158247142,0.598057501703323,-0.594384594525059],[0,0,0,0],[8.999999E+09,8.999999E+09,8.999999E+09,8.999999E+09,8.999999E+09,8.999999E+09]];
    LOCAL CONST Robtarget Tr_meulage_motif_1_148 := [[-42.891734375,61.9963046875,54.26795703125],[0.378981302219628,-0.381323158247142,0.598057501703323,-0.594384594525059],[0,0,0,0],[8.999999E+09,8.999999E+09,8.999999E+09,8.999999E+09,8.999999E+09,8.999999E+09]];
    LOCAL CONST Robtarget Tr_meulage_motif_1_149 := [[-42.667265625,62.44140625,53.1663359375],[0.378981302219628,-0.381323158247142,0.598057501703323,-0.594384594525059],[0,0,0,0],[8.999999E+09,8.999999E+09,8.999999E+09,8.999999E+09,8.999999E+09,8.999999E+09]];
    LOCAL CONST Robtarget Tr_meulage_motif_1_150 := [[-42.2939453125,63.212546875,52.1598203125],[0.378981302219628,-0.381323158247142,0.598057501703323,-0.594384594525059],[0,0,0,0],[8.999999E+09,8.999999E+09,8.999999E+09,8.999999E+09,8.999999E+09,8.999999E+09]];
    LOCAL CONST Robtarget Tr_meulage_motif_1_151 := [[-41.8532578125,64.13628515625,51.33103125],[0.378981302219628,-0.381323158247142,0.598057501703323,-0.594384594525059],[0,0,0,0],[8.999999E+09,8.999999E+09,8.999999E+09,8.999999E+09,8.999999E+09,8.999999E+09]];
    LOCAL CONST Robtarget Tr_meulage_motif_1_152 := [[-41.55967578125,64.7575234375,50.93531640625],[0.378981302219628,-0.381323158247142,0.598057501703323,-0.594384594525059],[0,0,0,0],[8.999999E+09,8.999999E+09,8.999999E+09,8.999999E+09,8.999999E+09,8.999999E+09]];
    LOCAL CONST Robtarget Tr_meulage_motif_1_153 := [[-41.06737109375,65.805859375,50.44782421875],[0.378981302219628,-0.381323158247142,0.598057501703323,-0.594384594525059],[0,0,0,0],[8.999999E+09,8.999999E+09,8.999999E+09,8.999999E+09,8.999999E+09,8.999999E+09]];
    LOCAL CONST Robtarget Tr_meulage_motif_1_154 := [[-40.70946875,66.571359375,50.18375],[0.378981302219628,-0.381323158247142,0.598057501703323,-0.594384594525059],[0,0,0,0],[8.999999E+09,8.999999E+09,8.999999E+09,8.999999E+09,8.999999E+09,8.999999E+09]];
    LOCAL CONST Robtarget Tr_meulage_motif_1_155 := [[-40.31596875,67.41621875,49.9792890625],[0.378981302219628,-0.381323158247142,0.598057501703323,-0.594384594525059],[0,0,0,0],[8.999999E+09,8.999999E+09,8.999999E+09,8.999999E+09,8.999999E+09,8.999999E+09]];
    LOCAL CONST Robtarget Tr_meulage_motif_1_156 := [[-39.9030625,68.3067109375,49.8706953125],[0.378981302219628,-0.381323158247142,0.598057501703323,-0.594384594525059],[0,0,0,0],[8.999999E+09,8.999999E+09,8.999999E+09,8.999999E+09,8.999999E+09,8.999999E+09]];
    LOCAL CONST Robtarget Tr_meulage_motif_1_157 := [[-39.485515625,69.207171875,49.76009765625],[0.378981302219628,-0.381323158247142,0.598057501703323,-0.594384594525059],[0,0,0,0],[8.999999E+09,8.999999E+09,8.999999E+09,8.999999E+09,8.999999E+09,8.999999E+09]];
    LOCAL CONST Robtarget Tr_meulage_motif_1_158 := [[-39.06642578125,70.1151171875,49.76008203125],[0.378981302219628,-0.381323158247142,0.598057501703323,-0.594384594525059],[0,0,0,0],[8.999999E+09,8.999999E+09,8.999999E+09,8.999999E+09,8.999999E+09,8.999999E+09]];
    LOCAL CONST Robtarget Tr_meulage_motif_1_159 := [[-38.6473359375,71.0230625,49.7600625],[0.378981302219628,-0.381323158247142,0.598057501703323,-0.594384594525059],[0,0,0,0],[8.999999E+09,8.999999E+09,8.999999E+09,8.999999E+09,8.999999E+09,8.999999E+09]];
    LOCAL CONST Robtarget Tr_meulage_motif_1_160 := [[-38.22824609375,71.9310078125,49.760046875],[0.378981302219628,-0.381323158247142,0.598057501703323,-0.594384594525059],[0,0,0,0],[8.999999E+09,8.999999E+09,8.999999E+09,8.999999E+09,8.999999E+09,8.999999E+09]];
    LOCAL CONST Robtarget Tr_meulage_motif_1_161 := [[-37.80915625,72.8389453125,49.76003125],[0.378981302219628,-0.381323158247142,0.598057501703323,-0.594384594525059],[0,0,0,0],[8.999999E+09,8.999999E+09,8.999999E+09,8.999999E+09,8.999999E+09,8.999999E+09]];
    LOCAL CONST Robtarget Tr_meulage_motif_1_162 := [[-37.39006640625,73.746890625,49.76001171875],[0.378981302219628,-0.381323158247142,0.598057501703323,-0.594384594525059],[0,0,0,0],[8.999999E+09,8.999999E+09,8.999999E+09,8.999999E+09,8.999999E+09,8.999999E+09]];
    LOCAL CONST Robtarget Tr_meulage_motif_1_163 := [[-36.9709765625,74.6548359375,49.75999609375],[0.378981302219628,-0.381323158247142,0.598057501703323,-0.594384594525059],[0,0,0,0],[8.999999E+09,8.999999E+09,8.999999E+09,8.999999E+09,8.999999E+09,8.999999E+09]];
    LOCAL CONST Robtarget Tr_meulage_motif_1_164 := [[-36.5518828125,75.56278125,49.75998046875],[0.378981302219628,-0.381323158247142,0.598057501703323,-0.594384594525059],[0,0,0,0],[8.999999E+09,8.999999E+09,8.999999E+09,8.999999E+09,8.999999E+09,8.999999E+09]];
    LOCAL CONST Robtarget Tr_meulage_motif_1_165 := [[-36.13279296875,76.4707265625,49.75996484375],[0.378981302219628,-0.381323158247142,0.598057501703323,-0.594384594525059],[0,0,0,0],[8.999999E+09,8.999999E+09,8.999999E+09,8.999999E+09,8.999999E+09,8.999999E+09]];
    LOCAL CONST Robtarget Tr_meulage_motif_1_166 := [[-35.713703125,77.378671875,49.7599453125],[0.378981302219628,-0.381323158247142,0.598057501703323,-0.594384594525059],[0,0,0,0],[8.999999E+09,8.999999E+09,8.999999E+09,8.999999E+09,8.999999E+09,8.999999E+09]];
    LOCAL CONST Robtarget Tr_meulage_motif_1_167 := [[-35.29461328125,78.2866171875,49.7599296875],[0.378981302219628,-0.381323158247142,0.598057501703323,-0.594384594525059],[0,0,0,0],[8.999999E+09,8.999999E+09,8.999999E+09,8.999999E+09,8.999999E+09,8.999999E+09]];
    LOCAL CONST Robtarget Tr_meulage_motif_1_168 := [[-34.8755234375,79.1945625,49.7599140625],[0.378981302219628,-0.381323158247142,0.598057501703323,-0.594384594525059],[0,0,0,0],[8.999999E+09,8.999999E+09,8.999999E+09,8.999999E+09,8.999999E+09,8.999999E+09]];
    LOCAL CONST Robtarget Tr_meulage_motif_1_169 := [[-34.45643359375,80.1025078125,49.75989453125],[0.378981302219628,-0.381323158247142,0.598057501703323,-0.594384594525059],[0,0,0,0],[8.999999E+09,8.999999E+09,8.999999E+09,8.999999E+09,8.999999E+09,8.999999E+09]];
    LOCAL CONST Robtarget Tr_meulage_motif_1_170 := [[-34.03734375,81.010453125,49.75987890625],[0.378981302219628,-0.381323158247142,0.598057501703323,-0.594384594525059],[0,0,0,0],[8.999999E+09,8.999999E+09,8.999999E+09,8.999999E+09,8.999999E+09,8.999999E+09]];
    LOCAL CONST Robtarget Tr_meulage_motif_1_171 := [[-33.61825390625,81.9183984375,49.75986328125],[0.378981302219628,-0.381323158247142,0.598057501703323,-0.594384594525059],[0,0,0,0],[8.999999E+09,8.999999E+09,8.999999E+09,8.999999E+09,8.999999E+09,8.999999E+09]];
    LOCAL CONST Robtarget Tr_meulage_motif_1_172 := [[-33.1991640625,82.8263359375,49.75984375],[0.378981302219628,-0.381323158247142,0.598057501703323,-0.594384594525059],[0,0,0,0],[8.999999E+09,8.999999E+09,8.999999E+09,8.999999E+09,8.999999E+09,8.999999E+09]];
    LOCAL CONST Robtarget Tr_meulage_motif_1_173 := [[-32.78007421875,83.73428125,49.759828125],[0.378981302219628,-0.381323158247142,0.598057501703323,-0.594384594525059],[0,0,0,0],[8.999999E+09,8.999999E+09,8.999999E+09,8.999999E+09,8.999999E+09,8.999999E+09]];
    LOCAL CONST Robtarget Tr_meulage_motif_1_174 := [[-32.360982421875,84.6422265625,49.7598125],[0.378981302219628,-0.381323158247142,0.598057501703323,-0.594384594525059],[0,0,0,0],[8.999999E+09,8.999999E+09,8.999999E+09,8.999999E+09,8.999999E+09,8.999999E+09]];
    LOCAL CONST Robtarget Tr_meulage_motif_1_175 := [[-31.941892578125,85.550171875,49.759796875],[0.378981302219628,-0.381323158247142,0.598057501703323,-0.594384594525059],[0,0,0,0],[8.999999E+09,8.999999E+09,8.999999E+09,8.999999E+09,8.999999E+09,8.999999E+09]];
    LOCAL CONST Robtarget Tr_meulage_motif_1_176 := [[-31.522802734375,86.4581171875,49.75977734375],[0.378981302219628,-0.381323158247142,0.598057501703323,-0.594384594525059],[0,0,0,0],[8.999999E+09,8.999999E+09,8.999999E+09,8.999999E+09,8.999999E+09,8.999999E+09]];
    LOCAL CONST Robtarget Tr_meulage_motif_1_177 := [[-31.1037109375,87.3660625,49.75976171875],[0.378981302219628,-0.381323158247142,0.598057501703323,-0.594384594525059],[0,0,0,0],[8.999999E+09,8.999999E+09,8.999999E+09,8.999999E+09,8.999999E+09,8.999999E+09]];
    LOCAL CONST Robtarget Tr_meulage_motif_1_178 := [[-30.68462109375,88.2740078125,49.75974609375],[0.378981302219628,-0.381323158247142,0.598057501703323,-0.594384594525059],[0,0,0,0],[8.999999E+09,8.999999E+09,8.999999E+09,8.999999E+09,8.999999E+09,8.999999E+09]];
    LOCAL CONST Robtarget Tr_meulage_motif_1_179 := [[-30.26553125,89.181953125,49.7597265625],[0.378981302219628,-0.381323158247142,0.598057501703323,-0.594384594525059],[0,0,0,0],[8.999999E+09,8.999999E+09,8.999999E+09,8.999999E+09,8.999999E+09,8.999999E+09]];
    LOCAL CONST Robtarget Tr_meulage_motif_1_180 := [[-29.84644140625,90.0898984375,49.7597109375],[0.378981302219628,-0.381323158247142,0.598057501703323,-0.594384594525059],[0,0,0,0],[8.999999E+09,8.999999E+09,8.999999E+09,8.999999E+09,8.999999E+09,8.999999E+09]];
    LOCAL CONST Robtarget Tr_meulage_motif_1_181 := [[-29.4273515625,90.99784375,49.7596953125],[0.378981302219628,-0.381323158247142,0.598057501703323,-0.594384594525059],[0,0,0,0],[8.999999E+09,8.999999E+09,8.999999E+09,8.999999E+09,8.999999E+09,8.999999E+09]];
    LOCAL CONST Robtarget Tr_meulage_motif_1_182 := [[-29.008259765625,91.9057890625,49.75967578125],[0.378981302219628,-0.381323158247142,0.598057501703323,-0.594384594525059],[0,0,0,0],[8.999999E+09,8.999999E+09,8.999999E+09,8.999999E+09,8.999999E+09,8.999999E+09]];
    LOCAL CONST Robtarget Tr_meulage_motif_1_183 := [[-28.589169921875,92.8137265625,49.75966015625],[0.378981302219628,-0.381323158247142,0.598057501703323,-0.594384594525059],[0,0,0,0],[8.999999E+09,8.999999E+09,8.999999E+09,8.999999E+09,8.999999E+09,8.999999E+09]];
    LOCAL CONST Robtarget Tr_meulage_motif_1_184 := [[-28.170080078125,93.721671875,49.75964453125],[0.378981302219628,-0.381323158247142,0.598057501703323,-0.594384594525059],[0,0,0,0],[8.999999E+09,8.999999E+09,8.999999E+09,8.999999E+09,8.999999E+09,8.999999E+09]];
    LOCAL CONST Robtarget Tr_meulage_motif_1_185 := [[-27.750990234375,94.6296171875,49.75962890625],[0.378981302219628,-0.381323158247142,0.598057501703323,-0.594384594525059],[0,0,0,0],[8.999999E+09,8.999999E+09,8.999999E+09,8.999999E+09,8.999999E+09,8.999999E+09]];
    LOCAL CONST Robtarget Tr_meulage_motif_1_186 := [[-27.331900390625,95.5375625,49.759609375],[0.378981302219628,-0.381323158247142,0.598057501703323,-0.594384594525059],[0,0,0,0],[8.999999E+09,8.999999E+09,8.999999E+09,8.999999E+09,8.999999E+09,8.999999E+09]];
    LOCAL CONST Robtarget Tr_meulage_motif_1_187 := [[-26.91280859375,96.4455078125,49.75959375],[0.378981302219628,-0.381323158247142,0.598057501703323,-0.594384594525059],[0,0,0,0],[8.999999E+09,8.999999E+09,8.999999E+09,8.999999E+09,8.999999E+09,8.999999E+09]];
    LOCAL CONST Robtarget Tr_meulage_motif_1_188 := [[-26.495263671875,97.34596875,49.64899609375],[0.378981302219628,-0.381323158247142,0.598057501703323,-0.594384594525059],[0,0,0,0],[8.999999E+09,8.999999E+09,8.999999E+09,8.999999E+09,8.999999E+09,8.999999E+09]];
    LOCAL CONST Robtarget Tr_meulage_motif_1_189 := [[-26.095591796875,98.203953125,49.4378203125],[0.378981302219628,-0.381323158247142,0.598057501703323,-0.594384594525059],[0,0,0,0],[8.999999E+09,8.999999E+09,8.999999E+09,8.999999E+09,8.999999E+09,8.999999E+09]];
    LOCAL CONST Robtarget Tr_meulage_motif_1_190 := [[-25.734359375,98.9763828125,49.16599609375],[0.378981302219628,-0.381323158247142,0.598057501703323,-0.594384594525059],[0,0,0,0],[8.999999E+09,8.999999E+09,8.999999E+09,8.999999E+09,8.999999E+09,8.999999E+09]];
    LOCAL CONST Robtarget Tr_meulage_motif_1_191 := [[-25.431849609375,99.6203828125,48.86187890625],[0.378981302219628,-0.381323158247142,0.598057501703323,-0.594384594525059],[0,0,0,0],[8.999999E+09,8.999999E+09,8.999999E+09,8.999999E+09,8.999999E+09,8.999999E+09]];
    LOCAL CONST Robtarget Tr_meulage_motif_1_192 := [[-24.988892578125,100.555265625,48.1994140625],[0.378981302219628,-0.381323158247142,0.598057501703323,-0.594384594525059],[0,0,0,0],[8.999999E+09,8.999999E+09,8.999999E+09,8.999999E+09,8.999999E+09,8.999999E+09]];
    LOCAL CONST Robtarget Tr_meulage_motif_1_193 := [[-24.598072265625,101.368234375,47.2975546875],[0.378981302219628,-0.381323158247142,0.598057501703323,-0.594384594525059],[0,0,0,0],[8.999999E+09,8.999999E+09,8.999999E+09,8.999999E+09,8.999999E+09,8.999999E+09]];
    LOCAL CONST Robtarget Tr_meulage_motif_1_194 := [[-24.35899609375,101.8470703125,46.25166015625],[0.378981302219628,-0.381323158247142,0.598057501703323,-0.594384594525059],[0,0,0,0],[8.999999E+09,8.999999E+09,8.999999E+09,8.999999E+09,8.999999E+09,8.999999E+09]];
    LOCAL CONST Robtarget Tr_meulage_motif_1_195 := [[-24.271697265625,102.01028125,45.5585078125],[0.378981302219628,-0.381323158247142,0.598057501703323,-0.594384594525059],[0,0,0,0],[8.999999E+09,8.999999E+09,8.999999E+09,8.999999E+09,8.999999E+09,8.999999E+09]];
    LOCAL CONST Robtarget Tr_meulage_motif_1_196 := [[-24.23398828125,102.063171875,44.7886015625],[0.378981302219628,-0.381323158247142,0.598057501703323,-0.594384594525059],[0,0,0,0],[8.999999E+09,8.999999E+09,8.999999E+09,8.999999E+09,8.999999E+09,8.999999E+09]];
    LOCAL CONST Robtarget Tr_meulage_motif_1_197 := [[-24.25109375,101.9973359375,44.0188359375],[0.378981302219628,-0.381323158247142,0.598057501703323,-0.594384594525059],[0,0,0,0],[8.999999E+09,8.999999E+09,8.999999E+09,8.999999E+09,8.999999E+09,8.999999E+09]];
    LOCAL CONST Robtarget Tr_meulage_motif_1_198 := [[-24.4111796875,101.6090703125,42.91073046875],[0.378981302219628,-0.381323158247142,0.598057501703323,-0.594384594525059],[0,0,0,0],[8.999999E+09,8.999999E+09,8.999999E+09,8.999999E+09,8.999999E+09,8.999999E+09]];
    LOCAL CONST Robtarget Tr_meulage_motif_1_199 := [[-24.576484375,101.2290390625,42.32512109375],[0.378981302219628,-0.381323158247142,0.598057501703323,-0.594384594525059],[0,0,0,0],[8.999999E+09,8.999999E+09,8.999999E+09,8.999999E+09,8.999999E+09,8.999999E+09]];
    LOCAL CONST Robtarget Tr_meulage_motif_1_200 := [[-24.93565234375,100.4177421875,41.43808984375],[0.378981302219628,-0.381323158247142,0.598057501703323,-0.594384594525059],[0,0,0,0],[8.999999E+09,8.999999E+09,8.999999E+09,8.999999E+09,8.999999E+09,8.999999E+09]];
    LOCAL CONST Robtarget Tr_meulage_motif_1_201 := [[-25.175216796875,99.8832421875,41.0238671875],[0.378981302219628,-0.381323158247142,0.598057501703323,-0.594384594525059],[0,0,0,0],[8.999999E+09,8.999999E+09,8.999999E+09,8.999999E+09,8.999999E+09,8.999999E+09]];
    LOCAL CONST Robtarget Tr_meulage_motif_1_202 := [[-25.635982421875,98.8646640625,40.479828125],[0.378981302219628,-0.381323158247142,0.598057501703323,-0.594384594525059],[0,0,0,0],[8.999999E+09,8.999999E+09,8.999999E+09,8.999999E+09,8.999999E+09,8.999999E+09]];
    LOCAL CONST Robtarget Tr_meulage_motif_1_203 := [[-25.97777734375,98.113125,40.18437890625],[0.378981302219628,-0.381323158247142,0.598057501703323,-0.594384594525059],[0,0,0,0],[8.999999E+09,8.999999E+09,8.999999E+09,8.999999E+09,8.999999E+09,8.999999E+09]];
    LOCAL CONST Robtarget Tr_meulage_motif_1_204 := [[-26.3654609375,97.2655703125,39.97993359375],[0.378981302219628,-0.381323158247142,0.598057501703323,-0.594384594525059],[0,0,0,0],[8.999999E+09,8.999999E+09,8.999999E+09,8.999999E+09,8.999999E+09,8.999999E+09]];
    LOCAL CONST Robtarget Tr_meulage_motif_1_205 := [[-26.77528125,96.37365625,39.87141796875],[0.378981302219628,-0.381323158247142,0.598057501703323,-0.594384594525059],[0,0,0,0],[8.999999E+09,8.999999E+09,8.999999E+09,8.999999E+09,8.999999E+09,8.999999E+09]];
    LOCAL CONST Robtarget Tr_meulage_motif_1_206 := [[-27.189681640625,95.471734375,39.76083984375],[0.378981302219628,-0.381323158247142,0.598057501703323,-0.594384594525059],[0,0,0,0],[8.999999E+09,8.999999E+09,8.999999E+09,8.999999E+09,8.999999E+09,8.999999E+09]];
    LOCAL CONST Robtarget Tr_meulage_motif_1_207 := [[-27.608771484375,94.5637890625,39.76085546875],[0.378981302219628,-0.381323158247142,0.598057501703323,-0.594384594525059],[0,0,0,0],[8.999999E+09,8.999999E+09,8.999999E+09,8.999999E+09,8.999999E+09,8.999999E+09]];
    LOCAL CONST Robtarget Tr_meulage_motif_1_208 := [[-28.027861328125,93.65584375,39.76087109375],[0.378981302219628,-0.381323158247142,0.598057501703323,-0.594384594525059],[0,0,0,0],[8.999999E+09,8.999999E+09,8.999999E+09,8.999999E+09,8.999999E+09,8.999999E+09]];
    LOCAL CONST Robtarget Tr_meulage_motif_1_209 := [[-28.446953125,92.7478984375,39.760890625],[0.378981302219628,-0.381323158247142,0.598057501703323,-0.594384594525059],[0,0,0,0],[8.999999E+09,8.999999E+09,8.999999E+09,8.999999E+09,8.999999E+09,8.999999E+09]];
    LOCAL CONST Robtarget Tr_meulage_motif_1_210 := [[-28.86604296875,91.839953125,39.76090625],[0.378981302219628,-0.381323158247142,0.598057501703323,-0.594384594525059],[0,0,0,0],[8.999999E+09,8.999999E+09,8.999999E+09,8.999999E+09,8.999999E+09,8.999999E+09]];
    LOCAL CONST Robtarget Tr_meulage_motif_1_211 := [[-29.2851328125,90.9320078125,39.760921875],[0.378981302219628,-0.381323158247142,0.598057501703323,-0.594384594525059],[0,0,0,0],[8.999999E+09,8.999999E+09,8.999999E+09,8.999999E+09,8.999999E+09,8.999999E+09]];
    LOCAL CONST Robtarget Tr_meulage_motif_1_212 := [[-29.70422265625,90.0240625,39.7609375],[0.378981302219628,-0.381323158247142,0.598057501703323,-0.594384594525059],[0,0,0,0],[8.999999E+09,8.999999E+09,8.999999E+09,8.999999E+09,8.999999E+09,8.999999E+09]];
    LOCAL CONST Robtarget Tr_meulage_motif_1_213 := [[-30.1233125,89.116125,39.76095703125],[0.378981302219628,-0.381323158247142,0.598057501703323,-0.594384594525059],[0,0,0,0],[8.999999E+09,8.999999E+09,8.999999E+09,8.999999E+09,8.999999E+09,8.999999E+09]];
    LOCAL CONST Robtarget Tr_meulage_motif_1_214 := [[-30.54240234375,88.2081796875,39.76097265625],[0.378981302219628,-0.381323158247142,0.598057501703323,-0.594384594525059],[0,0,0,0],[8.999999E+09,8.999999E+09,8.999999E+09,8.999999E+09,8.999999E+09,8.999999E+09]];
    LOCAL CONST Robtarget Tr_meulage_motif_1_215 := [[-30.961494140625,87.300234375,39.76098828125],[0.378981302219628,-0.381323158247142,0.598057501703323,-0.594384594525059],[0,0,0,0],[8.999999E+09,8.999999E+09,8.999999E+09,8.999999E+09,8.999999E+09,8.999999E+09]];
    LOCAL CONST Robtarget Tr_meulage_motif_1_216 := [[-31.380583984375,86.3922890625,39.7610078125],[0.378981302219628,-0.381323158247142,0.598057501703323,-0.594384594525059],[0,0,0,0],[8.999999E+09,8.999999E+09,8.999999E+09,8.999999E+09,8.999999E+09,8.999999E+09]];
    LOCAL CONST Robtarget Tr_meulage_motif_1_217 := [[-31.799673828125,85.48434375,39.7610234375],[0.378981302219628,-0.381323158247142,0.598057501703323,-0.594384594525059],[0,0,0,0],[8.999999E+09,8.999999E+09,8.999999E+09,8.999999E+09,8.999999E+09,8.999999E+09]];
    LOCAL CONST Robtarget Tr_meulage_motif_1_218 := [[-32.218763671875,84.5763984375,39.7610390625],[0.378981302219628,-0.381323158247142,0.598057501703323,-0.594384594525059],[0,0,0,0],[8.999999E+09,8.999999E+09,8.999999E+09,8.999999E+09,8.999999E+09,8.999999E+09]];
    LOCAL CONST Robtarget Tr_meulage_motif_1_219 := [[-32.637853515625,83.668453125,39.76105859375],[0.378981302219628,-0.381323158247142,0.598057501703323,-0.594384594525059],[0,0,0,0],[8.999999E+09,8.999999E+09,8.999999E+09,8.999999E+09,8.999999E+09,8.999999E+09]];
    LOCAL CONST Robtarget Tr_meulage_motif_1_220 := [[-33.0569453125,82.7605078125,39.76107421875],[0.378981302219628,-0.381323158247142,0.598057501703323,-0.594384594525059],[0,0,0,0],[8.999999E+09,8.999999E+09,8.999999E+09,8.999999E+09,8.999999E+09,8.999999E+09]];
    LOCAL CONST Robtarget Tr_meulage_motif_1_221 := [[-33.47603515625,81.8525625,39.76108984375],[0.378981302219628,-0.381323158247142,0.598057501703323,-0.594384594525059],[0,0,0,0],[8.999999E+09,8.999999E+09,8.999999E+09,8.999999E+09,8.999999E+09,8.999999E+09]];
    LOCAL CONST Robtarget Tr_meulage_motif_1_222 := [[-33.895125,80.9446171875,39.76110546875],[0.378981302219628,-0.381323158247142,0.598057501703323,-0.594384594525059],[0,0,0,0],[8.999999E+09,8.999999E+09,8.999999E+09,8.999999E+09,8.999999E+09,8.999999E+09]];
    LOCAL CONST Robtarget Tr_meulage_motif_1_223 := [[-34.31421484375,80.0366796875,39.761125],[0.378981302219628,-0.381323158247142,0.598057501703323,-0.594384594525059],[0,0,0,0],[8.999999E+09,8.999999E+09,8.999999E+09,8.999999E+09,8.999999E+09,8.999999E+09]];
    LOCAL CONST Robtarget Tr_meulage_motif_1_224 := [[-34.7333046875,79.128734375,39.761140625],[0.378981302219628,-0.381323158247142,0.598057501703323,-0.594384594525059],[0,0,0,0],[8.999999E+09,8.999999E+09,8.999999E+09,8.999999E+09,8.999999E+09,8.999999E+09]];
    LOCAL CONST Robtarget Tr_meulage_motif_1_225 := [[-35.15239453125,78.2207890625,39.76115625],[0.378981302219628,-0.381323158247142,0.598057501703323,-0.594384594525059],[0,0,0,0],[8.999999E+09,8.999999E+09,8.999999E+09,8.999999E+09,8.999999E+09,8.999999E+09]];
    LOCAL CONST Robtarget Tr_meulage_motif_1_226 := [[-35.571484375,77.31284375,39.76117578125],[0.378981302219628,-0.381323158247142,0.598057501703323,-0.594384594525059],[0,0,0,0],[8.999999E+09,8.999999E+09,8.999999E+09,8.999999E+09,8.999999E+09,8.999999E+09]];
    LOCAL CONST Robtarget Tr_meulage_motif_1_227 := [[-35.990578125,76.4048984375,39.76119140625],[0.378981302219628,-0.381323158247142,0.598057501703323,-0.594384594525059],[0,0,0,0],[8.999999E+09,8.999999E+09,8.999999E+09,8.999999E+09,8.999999E+09,8.999999E+09]];
    LOCAL CONST Robtarget Tr_meulage_motif_1_228 := [[-36.40966796875,75.496953125,39.76120703125],[0.378981302219628,-0.381323158247142,0.598057501703323,-0.594384594525059],[0,0,0,0],[8.999999E+09,8.999999E+09,8.999999E+09,8.999999E+09,8.999999E+09,8.999999E+09]];
    LOCAL CONST Robtarget Tr_meulage_motif_1_229 := [[-36.8287578125,74.5890078125,39.76122265625],[0.378981302219628,-0.381323158247142,0.598057501703323,-0.594384594525059],[0,0,0,0],[8.999999E+09,8.999999E+09,8.999999E+09,8.999999E+09,8.999999E+09,8.999999E+09]];
    LOCAL CONST Robtarget Tr_meulage_motif_1_230 := [[-37.24784765625,73.6810625,39.7612421875],[0.378981302219628,-0.381323158247142,0.598057501703323,-0.594384594525059],[0,0,0,0],[8.999999E+09,8.999999E+09,8.999999E+09,8.999999E+09,8.999999E+09,8.999999E+09]];
    LOCAL CONST Robtarget Tr_meulage_motif_1_231 := [[-37.6669375,72.7731171875,39.7612578125],[0.378981302219628,-0.381323158247142,0.598057501703323,-0.594384594525059],[0,0,0,0],[8.999999E+09,8.999999E+09,8.999999E+09,8.999999E+09,8.999999E+09,8.999999E+09]];
    LOCAL CONST Robtarget Tr_meulage_motif_1_232 := [[-38.08602734375,71.865171875,39.7612734375],[0.378981302219628,-0.381323158247142,0.598057501703323,-0.594384594525059],[0,0,0,0],[8.999999E+09,8.999999E+09,8.999999E+09,8.999999E+09,8.999999E+09,8.999999E+09]];
    LOCAL CONST Robtarget Tr_meulage_motif_1_233 := [[-38.5051171875,70.9572265625,39.76129296875],[0.378981302219628,-0.381323158247142,0.598057501703323,-0.594384594525059],[0,0,0,0],[8.999999E+09,8.999999E+09,8.999999E+09,8.999999E+09,8.999999E+09,8.999999E+09]];
    LOCAL CONST Robtarget Tr_meulage_motif_1_234 := [[-38.92420703125,70.0492890625,39.76130859375],[0.378981302219628,-0.381323158247142,0.598057501703323,-0.594384594525059],[0,0,0,0],[8.999999E+09,8.999999E+09,8.999999E+09,8.999999E+09,8.999999E+09,8.999999E+09]];
    LOCAL CONST Robtarget Tr_meulage_motif_1_235 := [[-39.343296875,69.14134375,39.76132421875],[0.378981302219628,-0.381323158247142,0.598057501703323,-0.594384594525059],[0,0,0,0],[8.999999E+09,8.999999E+09,8.999999E+09,8.999999E+09,8.999999E+09,8.999999E+09]];
    LOCAL CONST Robtarget Tr_meulage_motif_1_236 := [[-39.76238671875,68.2333984375,39.76134375],[0.378981302219628,-0.381323158247142,0.598057501703323,-0.594384594525059],[0,0,0,0],[8.999999E+09,8.999999E+09,8.999999E+09,8.999999E+09,8.999999E+09,8.999999E+09]];
    LOCAL CONST Robtarget Tr_meulage_motif_1_237 := [[-40.1767890625,67.3314765625,39.65076171875],[0.378981302219628,-0.381323158247142,0.598057501703323,-0.594384594525059],[0,0,0,0],[8.999999E+09,8.999999E+09,8.999999E+09,8.999999E+09,8.999999E+09,8.999999E+09]];
    LOCAL CONST Robtarget Tr_meulage_motif_1_238 := [[-40.570453125,66.47071875,39.4396171875],[0.378981302219628,-0.381323158247142,0.598057501703323,-0.594384594525059],[0,0,0,0],[8.999999E+09,8.999999E+09,8.999999E+09,8.999999E+09,8.999999E+09,8.999999E+09]];
    LOCAL CONST Robtarget Tr_meulage_motif_1_239 := [[-40.923953125,65.694703125,39.1678359375],[0.378981302219628,-0.381323158247142,0.598057501703323,-0.594384594525059],[0,0,0,0],[8.999999E+09,8.999999E+09,8.999999E+09,8.999999E+09,8.999999E+09,8.999999E+09]];
    LOCAL CONST Robtarget Tr_meulage_motif_1_240 := [[-41.2178125,65.04669921875,38.86374609375],[0.378981302219628,-0.381323158247142,0.598057501703323,-0.594384594525059],[0,0,0,0],[8.999999E+09,8.999999E+09,8.999999E+09,8.999999E+09,8.999999E+09,8.999999E+09]];
    LOCAL CONST Robtarget Tr_meulage_motif_1_241 := [[-41.64192578125,64.10309765625,38.2013125],[0.378981302219628,-0.381323158247142,0.598057501703323,-0.594384594525059],[0,0,0,0],[8.999999E+09,8.999999E+09,8.999999E+09,8.999999E+09,8.999999E+09,8.999999E+09]];
    LOCAL CONST Robtarget Tr_meulage_motif_1_242 := [[-41.9692265625,63.3588671875,37.26166015625],[0.378981302219628,-0.381323158247142,0.598057501703323,-0.594384594525059],[0,0,0,0],[8.999999E+09,8.999999E+09,8.999999E+09,8.999999E+09,8.999999E+09,8.999999E+09]];
    LOCAL CONST Robtarget Tr_meulage_motif_1_243 := [[-42.10276171875,63.0323125,36.2654296875],[0.378981302219628,-0.381323158247142,0.598057501703323,-0.594384594525059],[0,0,0,0],[8.999999E+09,8.999999E+09,8.999999E+09,8.999999E+09,8.999999E+09,8.999999E+09]];
    LOCAL CONST Robtarget Tr_meulage_motif_1_244 := [[-42.08240234375,63.0555703125,35.70794921875],[0.378981302219628,-0.381323158247142,0.598057501703323,-0.594384594525059],[0,0,0,0],[8.999999E+09,8.999999E+09,8.999999E+09,8.999999E+09,8.999999E+09,8.999999E+09]];
    LOCAL CONST Robtarget Tr_meulage_motif_1_245 := [[-42.078265625,63.04890234375,35.29009765625],[0.378981302219628,-0.381323158247142,0.598057501703323,-0.594384594525059],[0,0,0,0],[8.999999E+09,8.999999E+09,8.999999E+09,8.999999E+09,8.999999E+09,8.999999E+09]];
    LOCAL CONST Robtarget Tr_meulage_motif_1_246 := [[-41.912703125,63.37133984375,34.32087890625],[0.378981302219628,-0.381323158247142,0.598057501703323,-0.594384594525059],[0,0,0,0],[8.999999E+09,8.999999E+09,8.999999E+09,8.999999E+09,8.999999E+09,8.999999E+09]];
    LOCAL CONST Robtarget Tr_meulage_motif_1_247 := [[-41.5551875,64.11157421875,33.40329296875],[0.378981302219628,-0.381323158247142,0.598057501703323,-0.594384594525059],[0,0,0,0],[8.999999E+09,8.999999E+09,8.999999E+09,8.999999E+09,8.999999E+09,8.999999E+09]];
    LOCAL CONST Robtarget Tr_meulage_motif_1_248 := [[-41.292625,64.66459375,32.98044140625],[0.378981302219628,-0.381323158247142,0.598057501703323,-0.594384594525059],[0,0,0,0],[8.999999E+09,8.999999E+09,8.999999E+09,8.999999E+09,8.999999E+09,8.999999E+09]];
    LOCAL CONST Robtarget Tr_meulage_motif_1_249 := [[-40.81137890625,65.687359375,32.45003515625],[0.378981302219628,-0.381323158247142,0.598057501703323,-0.594384594525059],[0,0,0,0],[8.999999E+09,8.999999E+09,8.999999E+09,8.999999E+09,8.999999E+09,8.999999E+09]];
    LOCAL CONST Robtarget Tr_meulage_motif_1_250 := [[-40.4534765625,66.4528671875,32.1859453125],[0.378981302219628,-0.381323158247142,0.598057501703323,-0.594384594525059],[0,0,0,0],[8.999999E+09,8.999999E+09,8.999999E+09,8.999999E+09,8.999999E+09,8.999999E+09]];
    LOCAL CONST Robtarget Tr_meulage_motif_1_251 := [[-40.0599765625,67.2977265625,31.981470703125],[0.378981302219628,-0.381323158247142,0.598057501703323,-0.594384594525059],[0,0,0,0],[8.999999E+09,8.999999E+09,8.999999E+09,8.999999E+09,8.999999E+09,8.999999E+09]];
    LOCAL CONST Robtarget Tr_meulage_motif_1_252 := [[-39.6470703125,68.1882109375,31.872919921875],[0.378981302219628,-0.381323158247142,0.598057501703323,-0.594384594525059],[0,0,0,0],[8.999999E+09,8.999999E+09,8.999999E+09,8.999999E+09,8.999999E+09,8.999999E+09]];
    LOCAL CONST Robtarget Tr_meulage_motif_1_253 := [[-39.2295234375,69.0886796875,31.76230859375],[0.378981302219628,-0.381323158247142,0.598057501703323,-0.594384594525059],[0,0,0,0],[8.999999E+09,8.999999E+09,8.999999E+09,8.999999E+09,8.999999E+09,8.999999E+09]];
    LOCAL CONST Robtarget Tr_meulage_motif_1_254 := [[-38.81043359375,69.996625,31.762291015625],[0.378981302219628,-0.381323158247142,0.598057501703323,-0.594384594525059],[0,0,0,0],[8.999999E+09,8.999999E+09,8.999999E+09,8.999999E+09,8.999999E+09,8.999999E+09]];
    LOCAL CONST Robtarget Tr_meulage_motif_1_255 := [[-38.39134375,70.9045625,31.7622734375],[0.378981302219628,-0.381323158247142,0.598057501703323,-0.594384594525059],[0,0,0,0],[8.999999E+09,8.999999E+09,8.999999E+09,8.999999E+09,8.999999E+09,8.999999E+09]];
    LOCAL CONST Robtarget Tr_meulage_motif_1_256 := [[-37.97225390625,71.8125078125,31.7622578125],[0.378981302219628,-0.381323158247142,0.598057501703323,-0.594384594525059],[0,0,0,0],[8.999999E+09,8.999999E+09,8.999999E+09,8.999999E+09,8.999999E+09,8.999999E+09]];
    LOCAL CONST Robtarget Tr_meulage_motif_1_257 := [[-37.5531640625,72.720453125,31.762240234375],[0.378981302219628,-0.381323158247142,0.598057501703323,-0.594384594525059],[0,0,0,0],[8.999999E+09,8.999999E+09,8.999999E+09,8.999999E+09,8.999999E+09,8.999999E+09]];
    LOCAL CONST Robtarget Tr_meulage_motif_1_258 := [[-37.13407421875,73.6283984375,31.762224609375],[0.378981302219628,-0.381323158247142,0.598057501703323,-0.594384594525059],[0,0,0,0],[8.999999E+09,8.999999E+09,8.999999E+09,8.999999E+09,8.999999E+09,8.999999E+09]];
    LOCAL CONST Robtarget Tr_meulage_motif_1_259 := [[-36.71498046875,74.53634375,31.76220703125],[0.378981302219628,-0.381323158247142,0.598057501703323,-0.594384594525059],[0,0,0,0],[8.999999E+09,8.999999E+09,8.999999E+09,8.999999E+09,8.999999E+09,8.999999E+09]];
    LOCAL CONST Robtarget Tr_meulage_motif_1_260 := [[-36.295890625,75.4442890625,31.762189453125],[0.378981302219628,-0.381323158247142,0.598057501703323,-0.594384594525059],[0,0,0,0],[8.999999E+09,8.999999E+09,8.999999E+09,8.999999E+09,8.999999E+09,8.999999E+09]];
    LOCAL CONST Robtarget Tr_meulage_motif_1_261 := [[-35.87680078125,76.352234375,31.762173828125],[0.378981302219628,-0.381323158247142,0.598057501703323,-0.594384594525059],[0,0,0,0],[8.999999E+09,8.999999E+09,8.999999E+09,8.999999E+09,8.999999E+09,8.999999E+09]];
    LOCAL CONST Robtarget Tr_meulage_motif_1_262 := [[-35.4577109375,77.2601796875,31.76215625],[0.378981302219628,-0.381323158247142,0.598057501703323,-0.594384594525059],[0,0,0,0],[8.999999E+09,8.999999E+09,8.999999E+09,8.999999E+09,8.999999E+09,8.999999E+09]];
    LOCAL CONST Robtarget Tr_meulage_motif_1_263 := [[-35.03862109375,78.168125,31.762140625],[0.378981302219628,-0.381323158247142,0.598057501703323,-0.594384594525059],[0,0,0,0],[8.999999E+09,8.999999E+09,8.999999E+09,8.999999E+09,8.999999E+09,8.999999E+09]];
    LOCAL CONST Robtarget Tr_meulage_motif_1_264 := [[-34.61953125,79.0760703125,31.762123046875],[0.378981302219628,-0.381323158247142,0.598057501703323,-0.594384594525059],[0,0,0,0],[8.999999E+09,8.999999E+09,8.999999E+09,8.999999E+09,8.999999E+09,8.999999E+09]];
    LOCAL CONST Robtarget Tr_meulage_motif_1_265 := [[-34.20044140625,79.984015625,31.76210546875],[0.378981302219628,-0.381323158247142,0.598057501703323,-0.594384594525059],[0,0,0,0],[8.999999E+09,8.999999E+09,8.999999E+09,8.999999E+09,8.999999E+09,8.999999E+09]];
    LOCAL CONST Robtarget Tr_meulage_motif_1_266 := [[-33.7813515625,80.891953125,31.76208984375],[0.378981302219628,-0.381323158247142,0.598057501703323,-0.594384594525059],[0,0,0,0],[8.999999E+09,8.999999E+09,8.999999E+09,8.999999E+09,8.999999E+09,8.999999E+09]];
    LOCAL CONST Robtarget Tr_meulage_motif_1_267 := [[-33.36226171875,81.7998984375,31.762072265625],[0.378981302219628,-0.381323158247142,0.598057501703323,-0.594384594525059],[0,0,0,0],[8.999999E+09,8.999999E+09,8.999999E+09,8.999999E+09,8.999999E+09,8.999999E+09]];
    LOCAL CONST Robtarget Tr_meulage_motif_1_268 := [[-32.943171875,82.70784375,31.762056640625],[0.378981302219628,-0.381323158247142,0.598057501703323,-0.594384594525059],[0,0,0,0],[8.999999E+09,8.999999E+09,8.999999E+09,8.999999E+09,8.999999E+09,8.999999E+09]];
    LOCAL CONST Robtarget Tr_meulage_motif_1_269 := [[-32.524080078125,83.6157890625,31.7620390625],[0.378981302219628,-0.381323158247142,0.598057501703323,-0.594384594525059],[0,0,0,0],[8.999999E+09,8.999999E+09,8.999999E+09,8.999999E+09,8.999999E+09,8.999999E+09]];
    LOCAL CONST Robtarget Tr_meulage_motif_1_270 := [[-32.104990234375,84.523734375,31.762021484375],[0.378981302219628,-0.381323158247142,0.598057501703323,-0.594384594525059],[0,0,0,0],[8.999999E+09,8.999999E+09,8.999999E+09,8.999999E+09,8.999999E+09,8.999999E+09]];
    LOCAL CONST Robtarget Tr_meulage_motif_1_271 := [[-31.685900390625,85.4316796875,31.762005859375],[0.378981302219628,-0.381323158247142,0.598057501703323,-0.594384594525059],[0,0,0,0],[8.999999E+09,8.999999E+09,8.999999E+09,8.999999E+09,8.999999E+09,8.999999E+09]];
    LOCAL CONST Robtarget Tr_meulage_motif_1_272 := [[-31.26680859375,86.339625,31.76198828125],[0.378981302219628,-0.381323158247142,0.598057501703323,-0.594384594525059],[0,0,0,0],[8.999999E+09,8.999999E+09,8.999999E+09,8.999999E+09,8.999999E+09,8.999999E+09]];
    LOCAL CONST Robtarget Tr_meulage_motif_1_273 := [[-30.84771875,87.2475703125,31.76197265625],[0.378981302219628,-0.381323158247142,0.598057501703323,-0.594384594525059],[0,0,0,0],[8.999999E+09,8.999999E+09,8.999999E+09,8.999999E+09,8.999999E+09,8.999999E+09]];
    LOCAL CONST Robtarget Tr_meulage_motif_1_274 := [[-30.42862890625,88.155515625,31.761955078125],[0.378981302219628,-0.381323158247142,0.598057501703323,-0.594384594525059],[0,0,0,0],[8.999999E+09,8.999999E+09,8.999999E+09,8.999999E+09,8.999999E+09,8.999999E+09]];
    LOCAL CONST Robtarget Tr_meulage_motif_1_275 := [[-30.0095390625,89.0634609375,31.761939453125],[0.378981302219628,-0.381323158247142,0.598057501703323,-0.594384594525059],[0,0,0,0],[8.999999E+09,8.999999E+09,8.999999E+09,8.999999E+09,8.999999E+09,8.999999E+09]];
    LOCAL CONST Robtarget Tr_meulage_motif_1_276 := [[-29.59044921875,89.97140625,31.761921875],[0.378981302219628,-0.381323158247142,0.598057501703323,-0.594384594525059],[0,0,0,0],[8.999999E+09,8.999999E+09,8.999999E+09,8.999999E+09,8.999999E+09,8.999999E+09]];
    LOCAL CONST Robtarget Tr_meulage_motif_1_277 := [[-29.171357421875,90.87934375,31.761904296875],[0.378981302219628,-0.381323158247142,0.598057501703323,-0.594384594525059],[0,0,0,0],[8.999999E+09,8.999999E+09,8.999999E+09,8.999999E+09,8.999999E+09,8.999999E+09]];
    LOCAL CONST Robtarget Tr_meulage_motif_1_278 := [[-28.752267578125,91.7872890625,31.761888671875],[0.378981302219628,-0.381323158247142,0.598057501703323,-0.594384594525059],[0,0,0,0],[8.999999E+09,8.999999E+09,8.999999E+09,8.999999E+09,8.999999E+09,8.999999E+09]];
    LOCAL CONST Robtarget Tr_meulage_motif_1_279 := [[-28.333177734375,92.695234375,31.76187109375],[0.378981302219628,-0.381323158247142,0.598057501703323,-0.594384594525059],[0,0,0,0],[8.999999E+09,8.999999E+09,8.999999E+09,8.999999E+09,8.999999E+09,8.999999E+09]];
    LOCAL CONST Robtarget Tr_meulage_motif_1_280 := [[-27.914087890625,93.6031796875,31.76185546875],[0.378981302219628,-0.381323158247142,0.598057501703323,-0.594384594525059],[0,0,0,0],[8.999999E+09,8.999999E+09,8.999999E+09,8.999999E+09,8.999999E+09,8.999999E+09]];
    LOCAL CONST Robtarget Tr_meulage_motif_1_281 := [[-27.494998046875,94.511125,31.761837890625],[0.378981302219628,-0.381323158247142,0.598057501703323,-0.594384594525059],[0,0,0,0],[8.999999E+09,8.999999E+09,8.999999E+09,8.999999E+09,8.999999E+09,8.999999E+09]];
    LOCAL CONST Robtarget Tr_meulage_motif_1_282 := [[-27.07590625,95.4190703125,31.7618203125],[0.378981302219628,-0.381323158247142,0.598057501703323,-0.594384594525059],[0,0,0,0],[8.999999E+09,8.999999E+09,8.999999E+09,8.999999E+09,8.999999E+09,8.999999E+09]];
    LOCAL CONST Robtarget Tr_meulage_motif_1_283 := [[-26.65681640625,96.327015625,31.7618046875],[0.378981302219628,-0.381323158247142,0.598057501703323,-0.594384594525059],[0,0,0,0],[8.999999E+09,8.999999E+09,8.999999E+09,8.999999E+09,8.999999E+09,8.999999E+09]];
    LOCAL CONST Robtarget Tr_meulage_motif_1_284 := [[-26.2377265625,97.2349609375,31.761787109375],[0.378981302219628,-0.381323158247142,0.598057501703323,-0.594384594525059],[0,0,0,0],[8.999999E+09,8.999999E+09,8.999999E+09,8.999999E+09,8.999999E+09,8.999999E+09]];
    LOCAL CONST Robtarget Tr_meulage_motif_1_285 := [[-25.81863671875,98.14290625,31.761771484375],[0.378981302219628,-0.381323158247142,0.598057501703323,-0.594384594525059],[0,0,0,0],[8.999999E+09,8.999999E+09,8.999999E+09,8.999999E+09,8.999999E+09,8.999999E+09]];
    LOCAL CONST Robtarget Tr_meulage_motif_1_286 := [[-25.399546875,99.0508515625,31.76175390625],[0.378981302219628,-0.381323158247142,0.598057501703323,-0.594384594525059],[0,0,0,0],[8.999999E+09,8.999999E+09,8.999999E+09,8.999999E+09,8.999999E+09,8.999999E+09]];
    LOCAL CONST Robtarget Tr_meulage_motif_1_287 := [[-24.980455078125,99.9587890625,31.761736328125],[0.378981302219628,-0.381323158247142,0.598057501703323,-0.594384594525059],[0,0,0,0],[8.999999E+09,8.999999E+09,8.999999E+09,8.999999E+09,8.999999E+09,8.999999E+09]];
    LOCAL CONST Robtarget Tr_meulage_motif_1_288 := [[-24.561365234375,100.866734375,31.761720703125],[0.378981302219628,-0.381323158247142,0.598057501703323,-0.594384594525059],[0,0,0,0],[8.999999E+09,8.999999E+09,8.999999E+09,8.999999E+09,8.999999E+09,8.999999E+09]];
    LOCAL CONST Robtarget Tr_meulage_motif_1_289 := [[-24.142275390625,101.7746796875,31.761703125],[0.378981302219628,-0.381323158247142,0.598057501703323,-0.594384594525059],[0,0,0,0],[8.999999E+09,8.999999E+09,8.999999E+09,8.999999E+09,8.999999E+09,8.999999E+09]];
    LOCAL CONST Robtarget Tr_meulage_motif_1_290 := [[-23.723185546875,102.682625,31.7616875],[0.378981302219628,-0.381323158247142,0.598057501703323,-0.594384594525059],[0,0,0,0],[8.999999E+09,8.999999E+09,8.999999E+09,8.999999E+09,8.999999E+09,8.999999E+09]];
    LOCAL CONST Robtarget Tr_meulage_motif_1_291 := [[-23.304095703125,103.5905703125,31.761669921875],[0.378981302219628,-0.381323158247142,0.598057501703323,-0.594384594525059],[0,0,0,0],[8.999999E+09,8.999999E+09,8.999999E+09,8.999999E+09,8.999999E+09,8.999999E+09]];
    LOCAL CONST Robtarget Tr_meulage_motif_1_292 := [[-22.88500390625,104.498515625,31.761654296875],[0.378981302219628,-0.381323158247142,0.598057501703323,-0.594384594525059],[0,0,0,0],[8.999999E+09,8.999999E+09,8.999999E+09,8.999999E+09,8.999999E+09,8.999999E+09]];
    LOCAL CONST Robtarget Tr_meulage_motif_1_293 := [[-22.4659140625,105.4064609375,31.76163671875],[0.378981302219628,-0.381323158247142,0.598057501703323,-0.594384594525059],[0,0,0,0],[8.999999E+09,8.999999E+09,8.999999E+09,8.999999E+09,8.999999E+09,8.999999E+09]];
    LOCAL CONST Robtarget Tr_meulage_motif_1_294 := [[-22.04682421875,106.31440625,31.761619140625],[0.378981302219628,-0.381323158247142,0.598057501703323,-0.594384594525059],[0,0,0,0],[8.999999E+09,8.999999E+09,8.999999E+09,8.999999E+09,8.999999E+09,8.999999E+09]];

